LIN {X 0,Y 141.13,Z 751.048,A -85,B 0,C 180,E1 27006.176,E2 27006.176} C_VEL
LIN {X 0,Y 135.268,Z 754.68,A -85,B 0,C 180,E1 27012.954,E2 27012.954} C_VEL
LIN {X 0,Y 132.366,Z 756.637,A -85,B 0,C 180,E1 27014.356,E2 27014.356} C_VEL
LIN {X 0,Y 102.125,Z 773.9,A -85,B 0,C 180,E1 27021.98,E2 27021.98} C_VEL
LIN {X 0,Y 74.272,Z 785.098,A -85,B 0,C 180,E1 27035.392,E2 27035.392} C_VEL
LIN {X 0,Y 55.149,Z 790.593,A -85,B 0,C 180,E1 27056.715,E2 27056.715} C_VEL
LIN {X 0,Y 47.188,Z 792.386,A -85,B 0,C 180,E1 27090.017,E2 27090.017} C_VEL
LIN {X 0,Y 55.18,Z 790.549,A -85,B 0,C 180,E1 27123.299,E2 27123.299} C_VEL
LIN {X 0,Y 80.125,Z 782.969,A -85,B 0,C 180,E1 27148.264,E2 27148.264} C_VEL
LIN {X 0,Y 109.212,Z 770.247,A -85,B 0,C 180,E1 27160.115,E2 27160.115} C_VEL
LIN {X 0,Y 134.009,Z 755.358,A -85,B 0,C 180,E1 27165.896,E2 27165.896} C_VEL
LIN {X 0,Y 138.304,Z 752.387,A -85,B 0,C 180,E1 27170.176,E2 27170.176} C_VEL
LIN {X 0,Y 141.523,Z 750.747,A -85,B 0,C 180,E1 27175.02,E2 27175.02} C_VEL
LIN {X 0,Y 143.867,Z 750.723,A -85,B 0,C 180,E1 27180.669,E2 27180.669} C_VEL
LIN {X 0,Y 142.079,Z 752.687,A -85,B 0,C 180,E1 27182.028,E2 27182.028} C_VEL
LIN {X 0,Y 110.658,Z 774.445,A -85,B 0,C 180,E1 27187.223,E2 27187.223} C_VEL
LIN {X 0,Y 84.426,Z 788.358,A -85,B 0,C 180,E1 27195.358,E2 27195.358} C_VEL
LIN {X 0,Y 72.954,Z 792.741,A -85,B 0,C 180,E1 27198.842,E2 27198.842} C_VEL
LIN {X 0,Y 55.265,Z 797.756,A -85,B 0,C 180,E1 27205.481,E2 27205.481} C_VEL
LIN {X 0,Y 53.646,Z 798.256,A -85,B 0,C 180,E1 27206.938,E2 27206.938} C_VEL
LIN {X 0,Y 36.915,Z 804.117,A -85,B 0,C 180,E1 27245.763,E2 27245.763} C_VEL
LIN {X 0,Y 36.814,Z 805.147,A -85,B 0,C 180,E1 27269.978,E2 27269.978} C_VEL
LIN {X 0,Y 42.3,Z 802.077,A -85,B 0,C 180,E1 27315.686,E2 27315.686} C_VEL
LIN {X 0,Y 70.517,Z 792.25,A -85,B 0,C 180,E1 27345.009,E2 27345.009} C_VEL
LIN {X 0,Y 104.257,Z 776.595,A -85,B 0,C 180,E1 27355.878,E2 27355.878} C_VEL
LIN {X 0,Y 136.258,Z 756.023,A -85,B 0,C 180,E1 27360.693,E2 27360.693} C_VEL
LIN {X 0,Y 136.347,Z 755.474,A -85,B 0,C 180,E1 27362.184,E2 27362.184} C_VEL
LIN {X 0,Y 133.996,Z 756.111,A -85,B 0,C 180,E1 27366.506,E2 27366.506} C_VEL
LIN {X 0,Y 130.445,Z 758.02,A -85,B 0,C 180,E1 27370.436,E2 27370.436} C_VEL
LIN {X 0,Y 126.009,Z 760.827,A -85,B 0,C 180,E1 27371.835,E2 27371.835} C_VEL
LIN {X 0,Y 95.969,Z 776.64,A -85,B 0,C 180,E1 27378.841,E2 27378.841} C_VEL
LIN {X 0,Y 70.035,Z 786.286,A -85,B 0,C 180,E1 27390.172,E2 27390.172} C_VEL
LIN {X 0,Y 48.81,Z 791.778,A -85,B 0,C 180,E1 27411.678,E2 27411.678} C_VEL
LIN {X 0,Y 39.399,Z 793.569,A -85,B 0,C 180,E1 27450.02,E2 27450.02} C_VEL
LIN {X 0,Y 48.842,Z 791.735,A -85,B 0,C 180,E1 27488.334,E2 27488.334} C_VEL
LIN {X 0,Y 73.154,Z 785.238,A -85,B 0,C 180,E1 27511.616,E2 27511.616} C_VEL
LIN {X 0,Y 103.958,Z 772.802,A -85,B 0,C 180,E1 27523.35,E2 27523.35} C_VEL
LIN {X 0,Y 128.144,Z 759.249,A -85,B 0,C 180,E1 27528.457,E2 27528.457} C_VEL
LIN {X 0,Y 132.081,Z 756.912,A -85,B 0,C 180,E1 27531.11,E2 27531.11} C_VEL
LIN {X 0,Y 135.125,Z 755.518,A -85,B 0,C 180,E1 27535.552,E2 27535.552} C_VEL
LIN {X 0,Y 136.285,Z 755.805,A -85,B 0,C 180,E1 27539.325,E2 27539.325} C_VEL
LIN {X 0,Y 104.245,Z 776.442,A -85,B 0,C 180,E1 27544.079,E2 27544.079} C_VEL
LIN {X 0,Y 70.536,Z 792.156,A -85,B 0,C 180,E1 27554.96,E2 27554.96} C_VEL
LIN {X 0,Y 53.646,Z 798.256,A -85,B 0,C 180,E1 27566.938,E2 27566.938} C_VEL
LIN {X 0,Y 39.847,Z 801.381,A -85,B 0,C 180,E1 27579.711,E2 27579.711} C_VEL
LIN {X 0,Y 29.106,Z 803.028,A -85,B 0,C 180,E1 27603.278,E2 27603.278} C_VEL
LIN {X 0,Y 28.825,Z 803.933,A -85,B 0,C 180,E1 27629.972,E2 27629.972} C_VEL
LIN {X 0,Y 37.05,Z 800.835,A -85,B 0,C 180,E1 27684.776,E2 27684.776} C_VEL
LIN {X 0,Y 68.847,Z 790.999,A -85,B 0,C 180,E1 27711.647,E2 27711.647} C_VEL
LIN {X 0,Y 103.388,Z 775.666,A -85,B 0,C 180,E1 27720.281,E2 27720.281} C_VEL
LIN {X 0,Y 127.008,Z 761.504,A -85,B 0,C 180,E1 27723.22,E2 27723.22} C_VEL
LIN {X 0,Y 128.828,Z 760.178,A -85,B 0,C 180,E1 27723.807,E2 27723.807} C_VEL
LIN {X 0,Y 125.265,Z 761.647,A -85,B 0,C 180,E1 27728.171,E2 27728.171} C_VEL
LIN {X 0,Y 93.737,Z 777.832,A -85,B 0,C 180,E1 27734.315,E2 27734.315} C_VEL
LIN {X 0,Y 66.45,Z 787.475,A -85,B 0,C 180,E1 27744.334,E2 27744.334} C_VEL
LIN {X 0,Y 42.946,Z 792.966,A -85,B 0,C 180,E1 27765.19,E2 27765.19} C_VEL
LIN {X 0,Y 31.589,Z 794.756,A -85,B 0,C 180,E1 27810.025,E2 27810.025} C_VEL
LIN {X 0,Y 44.361,Z 792.68,A -85,B 0,C 180,E1 27856.879,E2 27856.879} C_VEL
LIN {X 0,Y 73.104,Z 785.355,A -85,B 0,C 180,E1 27878.774,E2 27878.774} C_VEL
LIN {X 0,Y 105.693,Z 772.261,A -85,B 0,C 180,E1 27888.307,E2 27888.307} C_VEL
LIN {X 0,Y 125.28,Z 761.436,A -85,B 0,C 180,E1 27891.786,E2 27891.786} C_VEL
LIN {X 0,Y 128.816,Z 759.994,A -85,B 0,C 180,E1 27896.178,E2 27896.178} C_VEL
LIN {X 0,Y 109.807,Z 771.944,A -85,B 0,C 180,E1 27898.744,E2 27898.744} C_VEL
LIN {X 0,Y 76.098,Z 788.137,A -85,B 0,C 180,E1 27905.75,E2 27905.75} C_VEL
LIN {X 0,Y 48.423,Z 797.618,A -85,B 0,C 180,E1 27920.311,E2 27920.311} C_VEL
LIN {X 0,Y 29.106,Z 803.028,A -85,B 0,C 180,E1 27963.278,E2 27963.278} C_VEL
LIN {X 0,Y 26.216,Z 803.383,A -85,B 0,C 180,E1 27980.281,E2 27980.281} C_VEL
LIN {X 0,Y 26.217,Z 800.978,A -85,B 0,C 180,E1 28042.764,E2 28042.764} C_VEL
LIN {X 0,Y 56.12,Z 793.66,A -85,B 0,C 180,E1 28074.433,E2 28074.433} C_VEL
LIN {X 0,Y 90.97,Z 780.586,A -85,B 0,C 180,E1 28083.207,E2 28083.207} C_VEL
LIN {X 0,Y 113.201,Z 769.259,A -85,B 0,C 180,E1 28085.73,E2 28085.73} C_VEL
LIN {X 0,Y 81.265,Z 783.16,A -85,B 0,C 180,E1 28092.058,E2 28092.058} C_VEL
LIN {X 0,Y 50.114,Z 791.904,A -85,B 0,C 180,E1 28105.032,E2 28105.032} C_VEL
LIN {X 0,Y 28.183,Z 795.415,A -85,B 0,C 180,E1 28137.54,E2 28137.54} C_VEL
LIN {X 0,Y 28.206,Z 795.39,A -85,B 0,C 180,E1 28202.498,E2 28202.498} C_VEL
LIN {X 0,Y 56.821,Z 790.364,A -85,B 0,C 180,E1 28238.881,E2 28238.881} C_VEL
LIN {X 0,Y 88.526,Z 780.33,A -85,B 0,C 180,E1 28249.594,E2 28249.594} C_VEL
LIN {X 0,Y 113.197,Z 769.09,A -85,B 0,C 180,E1 28254.216,E2 28254.216} C_VEL
LIN {X 0,Y 79.519,Z 785.367,A -85,B 0,C 180,E1 28258.743,E2 28258.743} C_VEL
LIN {X 0,Y 46.237,Z 796.364,A -85,B 0,C 180,E1 28270.691,E2 28270.691} C_VEL
LIN {X 0,Y 21.523,Z 801.927,A -85,B 0,C 180,E1 28318.32,E2 28318.32} C_VEL
LIN {X 0,Y 20.825,Z 802.718,A -85,B 0,C 180,E1 28349.962,E2 28349.962} C_VEL
LIN {X 0,Y 26.217,Z 800.978,A -85,B 0,C 180,E1 28402.764,E2 28402.764} C_VEL
LIN {X 0,Y 33.884,Z 798.843,A -85,B 0,C 180,E1 28422.95,E2 28422.95} C_VEL
LIN {X 0,Y 48.682,Z 794.374,A -85,B 0,C 180,E1 28440.59,E2 28440.59} C_VEL
LIN {X 0,Y 50.712,Z 793.84,A -85,B 0,C 180,E1 28441.362,E2 28441.362} C_VEL
LIN {X 0,Y 76.198,Z 785.741,A -85,B 0,C 180,E1 28446.637,E2 28446.637} C_VEL
LIN {X 0,Y 76.303,Z 785.609,A -85,B 0,C 180,E1 28447.283,E2 28447.283} C_VEL
LIN {X 0,Y 47.344,Z 793.089,A -85,B 0,C 180,E1 28456.449,E2 28456.449} C_VEL
LIN {X 0,Y 22.001,Z 796.601,A -85,B 0,C 180,E1 28486.566,E2 28486.566} C_VEL
LIN {X 0,Y 22.027,Z 796.576,A -85,B 0,C 180,E1 28573.47,E2 28573.47} C_VEL
LIN {X 0,Y 54.647,Z 791.518,A -85,B 0,C 180,E1 28606.631,E2 28606.631} C_VEL
LIN {X 0,Y 76.341,Z 785.486,A -85,B 0,C 180,E1 28612.66,E2 28612.66} C_VEL
LIN {X 0,Y 73.357,Z 786.71,A -85,B 0,C 180,E1 28613.712,E2 28613.712} C_VEL
LIN {X 0,Y 37.959,Z 796.821,A -85,B 0,C 180,E1 28624.055,E2 28624.055} C_VEL
LIN {X 0,Y 17.803,Z 800.424,A -85,B 0,C 180,E1 28651.658,E2 28651.658} C_VEL
LIN {X 0,Y 12.836,Z 801.505,A -85,B 0,C 180,E1 28709.938,E2 28709.938} C_VEL
LIN {X 0,Y 30.675,Z 798.349,A -85,B 0,C 180,E1 28790.64,E2 28790.64} C_VEL
LIN {X 0,Y 50.712,Z 793.84,A -85,B 0,C 180,E1 28801.362,E2 28801.362} C_VEL
LIN {X 0,Y 47.229,Z 794.189,A -85,B 0,C 180,E1 28805.113,E2 28805.113} C_VEL
LIN {X 0,Y 18.1,Z 797.697,A -85,B 0,C 180,E1 28826.556,E2 28826.556} C_VEL
LIN {X 0,Y 17.221,Z 797.762,A -85,B 0,C 180,E1 28951.638,E2 28951.638} C_VEL
LIN {X 0,Y 31.108,Z 796.48,A -85,B 0,C 180,E1 28966.867,E2 28966.867} C_VEL
LIN {X 0,Y 36.979,Z 795.832,A -85,B 0,C 180,E1 28971.997,E2 28971.997} C_VEL
LIN {X 0,Y 15.203,Z 799.19,A -85,B 0,C 180,E1 28984.607,E2 28984.607} C_VEL
LIN {X 0,Y 4.811,Z 800.285,A -85,B 0,C 180,E1 29069.834,E2 29069.834} C_VEL
LIN {X 0,Y 30.434,Z 797.108,A -85,B 0,C 180,E1 29166.009,E2 29166.009} C_VEL
LIN {X 0,Y 36.911,Z 795.896,A -85,B 0,C 180,E1 29167.955,E2 29167.955} C_VEL
LIN {X 0,Y 31.072,Z 796.524,A -85,B 0,C 180,E1 29173.079,E2 29173.079} C_VEL
LIN {X 0,Y 18.1,Z 797.697,A -85,B 0,C 180,E1 29186.556,E2 29186.556} C_VEL
LIN {X 0,Y 16.552,Z 799.69,A -85,B 0,C 180,E1 29189.815,E2 29189.815} C_VEL
LIN {X 0,Y 16.552,Z 875,A -85,B 0,C 180,E1 29189.815,E2 29189.815} C_VEL
LIN {X 0,Y 16.552,Z 875,A -85,B 0,C 180,E1 29189.815,E2 29189.815}

QRS_NEXT_CUT()
PTP {E1 29336.944,E2 29336.944}
PTP {X 0,Y 607.85,A -85,B 0,C 180,E1 29336.944,E2 29336.944,E3 0,E4 0,E5 0,E6 0}
QRS_SPEED_INIT()
LIN {X 0,Y 607.85,Z 875,A -85,B 0,C 180,E1 29336.944,E2 29336.944,E3 0,E4 0,E5 0,E6 0} C_VEL
LIN {X 0,Y 607.85,Z 296.842,A -85,B 0,C 180,E1 29336.944,E2 29336.944} C_VEL
LIN {X 0,Y 607.85,Z 288.764,A -85,B 0,C 180,E1 29336.944,E2 29336.944} C_VEL
LIN {X 0,Y 607.871,Z 286.764,A -85,B 0,C 180,E1 29336.755,E2 29336.755} C_VEL
LIN {X 0,Y 607.835,Z 286.764,A -85,B 0,C 180,E1 29333.672,E2 29333.672} C_VEL
LIN {X 0,Y 607.851,Z 286.764,A -85,B 0,C 180,E1 29330.914,E2 29330.914} C_VEL
LIN {X 0,Y 607.842,Z 286.764,A -85,B 0,C 180,E1 29327.652,E2 29327.652} C_VEL
LIN {X 0,Y 607.86,Z 286.764,A -85,B 0,C 180,E1 29324.839,E2 29324.839} C_VEL
LIN {X 0,Y 607.85,Z 286.762,A -85,B 0,C 180,E1 29321.589,E2 29321.589} C_VEL
LIN {X 0,Y 607.875,Z 286.764,A -85,B 0,C 180,E1 29318.684,E2 29318.684} C_VEL
LIN {X 0,Y 607.856,Z 286.761,A -85,B 0,C 180,E1 29315.511,E2 29315.511} C_VEL
LIN {X 0,Y 607.886,Z 286.764,A -85,B 0,C 180,E1 29312.577,E2 29312.577} C_VEL
LIN {X 0,Y 607.862,Z 286.761,A -85,B 0,C 180,E1 29309.451,E2 29309.451} C_VEL
LIN {X 0,Y 607.899,Z 286.764,A -85,B 0,C 180,E1 29306.451,E2 29306.451} C_VEL
LIN {X 0,Y 607.865,Z 286.76,A -85,B 0,C 180,E1 29303.338,E2 29303.338} C_VEL
LIN {X 0,Y 607.909,Z 286.765,A -85,B 0,C 180,E1 29300.329,E2 29300.329} C_VEL
LIN {X 0,Y 607.867,Z 286.76,A -85,B 0,C 180,E1 29297.188,E2 29297.188} C_VEL
LIN {X 0,Y 607.915,Z 286.761,A -85,B 0,C 180,E1 29294.083,E2 29294.083} C_VEL
LIN {X 0,Y 607.87,Z 286.76,A -85,B 0,C 180,E1 29290.975,E2 29290.975} C_VEL
LIN {X 0,Y 607.912,Z 286.759,A -85,B 0,C 180,E1 29287.841,E2 29287.841} C_VEL
LIN {X 0,Y 607.879,Z 286.761,A -85,B 0,C 180,E1 29284.687,E2 29284.687} C_VEL
LIN {X 0,Y 607.911,Z 286.755,A -85,B 0,C 180,E1 29281.535,E2 29281.535} C_VEL
LIN {X 0,Y 607.905,Z 286.765,A -85,B 0,C 180,E1 29278.273,E2 29278.273} C_VEL
LIN {X 0,Y 607.909,Z 287.028,A -85,B 0,C 180,E1 29276.259,E2 29276.259} C_VEL
LIN {X 0,Y 607.912,Z 319.926,A -85,B 0,C 180,E1 29273.454,E2 29273.454} C_VEL
LIN {X 0,Y 607.914,Z 334.281,A -85,B 0,C 180,E1 29272.278,E2 29272.278} C_VEL
LIN {X 0,Y 607.916,Z 541.958,A -85,B 0,C 180,E1 29269.666,E2 29269.666} C_VEL
LIN {X 0,Y 607.911,Z 560.928,A -85,B 0,C 180,E1 29269.25,E2 29269.25} C_VEL
LIN {X 0,Y 607.902,Z 579.266,A -85,B 0,C 180,E1 29268.668,E2 29268.668} C_VEL
LIN {X 0,Y 607.897,Z 597.163,A -85,B 0,C 180,E1 29267.913,E2 29267.913} C_VEL
LIN {X 0,Y 607.919,Z 613.869,A -85,B 0,C 180,E1 29267.023,E2 29267.023} C_VEL
LIN {X 0,Y 607.917,Z 629.704,A -85,B 0,C 180,E1 29265.991,E2 29265.991} C_VEL
LIN {X 0,Y 607.917,Z 644.611,A -85,B 0,C 180,E1 29264.818,E2 29264.818} C_VEL
LIN {X 0,Y 607.915,Z 658.52,A -85,B 0,C 180,E1 29263.506,E2 29263.506} C_VEL
LIN {X 0,Y 607.917,Z 671.323,A -85,B 0,C 180,E1 29262.056,E2 29262.056} C_VEL
LIN {X 0,Y 607.911,Z 682.566,A -85,B 0,C 180,E1 29260.519,E2 29260.519} C_VEL
LIN {X 0,Y 607.914,Z 692.264,A -85,B 0,C 180,E1 29258.894,E2 29258.894} C_VEL
LIN {X 0,Y 607.911,Z 699.987,A -85,B 0,C 180,E1 29257.276,E2 29257.276} C_VEL
LIN {X 0,Y 607.907,Z 706.267,A -85,B 0,C 180,E1 29255.569,E2 29255.569} C_VEL
LIN {X 0,Y 607.918,Z 710.775,A -85,B 0,C 180,E1 29253.867,E2 29253.867} C_VEL
LIN {X 0,Y 607.917,Z 713.734,A -85,B 0,C 180,E1 29252.074,E2 29252.074} C_VEL
LIN {X 0,Y 607.908,Z 714.929,A -85,B 0,C 180,E1 29250.283,E2 29250.283} C_VEL
LIN {X 0,Y 607.915,Z 714.38,A -85,B 0,C 180,E1 29248.492,E2 29248.492} C_VEL
LIN {X 0,Y 607.909,Z 712.08,A -85,B 0,C 180,E1 29246.7,E2 29246.7} C_VEL
LIN {X 0,Y 607.914,Z 708.217,A -85,B 0,C 180,E1 29244.999,E2 29244.999} C_VEL
LIN {X 0,Y 607.91,Z 702.635,A -85,B 0,C 180,E1 29243.294,E2 29243.294} C_VEL
LIN {X 0,Y 607.917,Z 695.641,A -85,B 0,C 180,E1 29241.678,E2 29241.678} C_VEL
LIN {X 0,Y 607.913,Z 686.781,A -85,B 0,C 180,E1 29240.056,E2 29240.056} C_VEL
LIN {X 0,Y 607.917,Z 676.477,A -85,B 0,C 180,E1 29238.521,E2 29238.521} C_VEL
LIN {X 0,Y 607.913,Z 664.743,A -85,B 0,C 180,E1 29237.075,E2 29237.075} C_VEL
LIN {X 0,Y 607.917,Z 651.561,A -85,B 0,C 180,E1 29235.718,E2 29235.718} C_VEL
LIN {X 0,Y 607.917,Z 636.801,A -85,B 0,C 180,E1 29234.45,E2 29234.45} C_VEL
LIN {X 0,Y 607.917,Z 620.944,A -85,B 0,C 180,E1 29233.322,E2 29233.322} C_VEL
LIN {X 0,Y 607.902,Z 603.949,A -85,B 0,C 180,E1 29232.335,E2 29232.335} C_VEL
LIN {X 0,Y 607.918,Z 586.961,A -85,B 0,C 180,E1 29231.543,E2 29231.543} C_VEL
LIN {X 0,Y 607.909,Z 569.084,A -85,B 0,C 180,E1 29230.895,E2 29230.895} C_VEL
LIN {X 0,Y 607.915,Z 550.763,A -85,B 0,C 180,E1 29230.413,E2 29230.413} C_VEL
LIN {X 0,Y 607.918,Z 531.813,A -85,B 0,C 180,E1 29230.096,E2 29230.096} C_VEL
LIN {X 0,Y 607.91,Z 334.059,A -85,B 0,C 180,E1 29227.621,E2 29227.621} C_VEL
LIN {X 0,Y 607.918,Z 296.429,A -85,B 0,C 180,E1 29224.475,E2 29224.475} C_VEL
LIN {X 0,Y 607.909,Z 286.947,A -85,B 0,C 180,E1 29223.636,E2 29223.636} C_VEL
LIN {X 0,Y 607.91,Z 286.756,A -85,B 0,C 180,E1 29220.543,E2 29220.543} C_VEL
LIN {X 0,Y 607.889,Z 286.762,A -85,B 0,C 180,E1 29217.352,E2 29217.352} C_VEL
LIN {X 0,Y 607.91,Z 286.758,A -85,B 0,C 180,E1 29214.181,E2 29214.181} C_VEL
LIN {X 0,Y 607.877,Z 286.76,A -85,B 0,C 180,E1 29211.075,E2 29211.075} C_VEL
LIN {X 0,Y 607.91,Z 286.76,A -85,B 0,C 180,E1 29207.98,E2 29207.98} C_VEL
LIN {X 0,Y 607.872,Z 286.759,A -85,B 0,C 180,E1 29204.882,E2 29204.882} C_VEL
LIN {X 0,Y 607.918,Z 286.764,A -85,B 0,C 180,E1 29201.696,E2 29201.696} C_VEL
LIN {X 0,Y 607.877,Z 286.759,A -85,B 0,C 180,E1 29198.565,E2 29198.565} C_VEL
LIN {X 0,Y 607.879,Z 286.763,A -85,B 0,C 180,E1 29195.264,E2 29195.264} C_VEL
LIN {X 0,Y 607.897,Z 286.758,A -85,B 0,C 180,E1 29192.203,E2 29192.203} C_VEL
LIN {X 0,Y 607.862,Z 286.762,A -85,B 0,C 180,E1 29189.028,E2 29189.028} C_VEL
LIN {X 0,Y 607.903,Z 286.759,A -85,B 0,C 180,E1 29186.05,E2 29186.05} C_VEL
LIN {X 0,Y 607.854,Z 286.763,A -85,B 0,C 180,E1 29182.91,E2 29182.91} C_VEL
LIN {X 0,Y 607.905,Z 286.76,A -85,B 0,C 180,E1 29179.905,E2 29179.905} C_VEL
LIN {X 0,Y 607.846,Z 286.763,A -85,B 0,C 180,E1 29176.801,E2 29176.801} C_VEL
LIN {X 0,Y 607.909,Z 286.761,A -85,B 0,C 180,E1 29173.798,E2 29173.798} C_VEL
LIN {X 0,Y 607.839,Z 286.764,A -85,B 0,C 180,E1 29170.713,E2 29170.713} C_VEL
LIN {X 0,Y 607.899,Z 286.762,A -85,B 0,C 180,E1 29167.751,E2 29167.751} C_VEL
LIN {X 0,Y 607.834,Z 286.764,A -85,B 0,C 180,E1 29164.718,E2 29164.718} C_VEL
LIN {X 0,Y 607.866,Z 286.764,A -85,B 0,C 180,E1 29161.885,E2 29161.885} C_VEL
LIN {X 0,Y 607.834,Z 286.765,A -85,B 0,C 180,E1 29158.775,E2 29158.775} C_VEL
LIN {X 0,Y 607.846,Z 286.764,A -85,B 0,C 180,E1 29156.039,E2 29156.039} C_VEL
LIN {X 0,Y 607.848,Z 286.763,A -85,B 0,C 180,E1 29152.819,E2 29152.819} C_VEL
LIN {X 0,Y 607.847,Z 286.764,A -85,B 0,C 180,E1 29150.054,E2 29150.054} C_VEL
LIN {X 0,Y 607.857,Z 286.762,A -85,B 0,C 180,E1 29146.783,E2 29146.783} C_VEL
LIN {X 0,Y 607.856,Z 286.764,A -85,B 0,C 180,E1 29143.958,E2 29143.958} C_VEL
LIN {X 0,Y 607.861,Z 286.761,A -85,B 0,C 180,E1 29140.694,E2 29140.694} C_VEL
LIN {X 0,Y 607.873,Z 286.764,A -85,B 0,C 180,E1 29137.771,E2 29137.771} C_VEL
LIN {X 0,Y 607.862,Z 286.761,A -85,B 0,C 180,E1 29134.557,E2 29134.557} C_VEL
LIN {X 0,Y 607.889,Z 286.764,A -85,B 0,C 180,E1 29131.618,E2 29131.618} C_VEL
LIN {X 0,Y 607.865,Z 286.76,A -85,B 0,C 180,E1 29128.432,E2 29128.432} C_VEL
LIN {X 0,Y 607.918,Z 286.763,A -85,B 0,C 180,E1 29125.314,E2 29125.314} C_VEL
LIN {X 0,Y 607.867,Z 286.76,A -85,B 0,C 180,E1 29122.274,E2 29122.274} C_VEL
LIN {X 0,Y 607.914,Z 286.761,A -85,B 0,C 180,E1 29119.162,E2 29119.162} C_VEL
LIN {X 0,Y 607.871,Z 286.76,A -85,B 0,C 180,E1 29116.042,E2 29116.042} C_VEL
LIN {X 0,Y 607.913,Z 286.759,A -85,B 0,C 180,E1 29112.914,E2 29112.914} C_VEL
LIN {X 0,Y 607.88,Z 286.761,A -85,B 0,C 180,E1 29109.778,E2 29109.778} C_VEL
LIN {X 0,Y 607.908,Z 286.756,A -85,B 0,C 180,E1 29106.54,E2 29106.54} C_VEL
LIN {X 0,Y 607.897,Z 286.884,A -85,B 0,C 180,E1 29103.498,E2 29103.498} C_VEL
LIN {X 0,Y 607.908,Z 287.709,A -85,B 0,C 180,E1 29103.382,E2 29103.382} C_VEL
LIN {X 0,Y 607.913,Z 340.141,A -85,B 0,C 180,E1 29100.435,E2 29100.435} C_VEL
LIN {X 0,Y 607.885,Z 390.509,A -85,B 0,C 180,E1 29097.701,E2 29097.701} C_VEL
LIN {X 0,Y 607.913,Z 616.116,A -85,B 0,C 180,E1 29094.784,E2 29094.784} C_VEL
LIN {X 0,Y 607.918,Z 653.733,A -85,B 0,C 180,E1 29094.278,E2 29094.278} C_VEL
LIN {X 0,Y 607.906,Z 673.698,A -85,B 0,C 180,E1 29093.84,E2 29093.84} C_VEL
LIN {X 0,Y 607.911,Z 693.06,A -85,B 0,C 180,E1 29093.249,E2 29093.249} C_VEL
LIN {X 0,Y 607.915,Z 712.501,A -85,B 0,C 180,E1 29092.482,E2 29092.482} C_VEL
LIN {X 0,Y 607.919,Z 731.168,A -85,B 0,C 180,E1 29091.567,E2 29091.567} C_VEL
LIN {X 0,Y 607.917,Z 749.766,A -85,B 0,C 180,E1 29090.456,E2 29090.456} C_VEL
LIN {X 0,Y 607.913,Z 767.254,A -85,B 0,C 180,E1 29089.204,E2 29089.204} C_VEL
LIN {X 0,Y 607.911,Z 783.162,A -85,B 0,C 180,E1 29087.863,E2 29087.863} C_VEL
LIN {X 0,Y 607.915,Z 797.673,A -85,B 0,C 180,E1 29086.432,E2 29086.432} C_VEL
LIN {X 0,Y 607.909,Z 811.263,A -85,B 0,C 180,E1 29084.867,E2 29084.867} C_VEL
LIN {X 0,Y 607.918,Z 823.719,A -85,B 0,C 180,E1 29083.176,E2 29083.176} C_VEL
LIN {X 0,Y 607.906,Z 834.252,A -85,B 0,C 180,E1 29081.479,E2 29081.479} C_VEL
LIN {X 0,Y 607.907,Z 843.561,A -85,B 0,C 180,E1 29079.658,E2 29079.658} C_VEL
LIN {X 0,Y 607.907,Z 850.973,A -85,B 0,C 180,E1 29077.846,E2 29077.846} C_VEL
LIN {X 0,Y 607.913,Z 856.989,A -85,B 0,C 180,E1 29075.947,E2 29075.947} C_VEL
LIN {X 0,Y 607.913,Z 861.292,A -85,B 0,C 180,E1 29074.055,E2 29074.055} C_VEL
LIN {X 0,Y 607.909,Z 863.95,A -85,B 0,C 180,E1 29072.168,E2 29072.168} C_VEL
LIN {X 0,Y 607.902,Z 864.94,A -85,B 0,C 180,E1 29070.283,E2 29070.283} C_VEL
LIN {X 0,Y 607.904,Z 864.372,A -85,B 0,C 180,E1 29068.398,E2 29068.398} C_VEL
LIN {X 0,Y 607.908,Z 862.082,A -85,B 0,C 180,E1 29066.417,E2 29066.417} C_VEL
LIN {X 0,Y 607.91,Z 858.255,A -85,B 0,C 180,E1 29064.526,E2 29064.526} C_VEL
LIN {X 0,Y 607.913,Z 852.689,A -85,B 0,C 180,E1 29062.629,E2 29062.629} C_VEL
LIN {X 0,Y 607.919,Z 845.655,A -85,B 0,C 180,E1 29060.82,E2 29060.82} C_VEL
LIN {X 0,Y 607.909,Z 836.843,A -85,B 0,C 180,E1 29059.001,E2 29059.001} C_VEL
LIN {X 0,Y 607.911,Z 826.516,A -85,B 0,C 180,E1 29057.247,E2 29057.247} C_VEL
LIN {X 0,Y 607.917,Z 815.136,A -85,B 0,C 180,E1 29055.62,E2 29055.62} C_VEL
LIN {X 0,Y 607.91,Z 801.355,A -85,B 0,C 180,E1 29053.96,E2 29053.96} C_VEL
LIN {X 0,Y 607.918,Z 785.904,A -85,B 0,C 180,E1 29052.385,E2 29052.385} C_VEL
LIN {X 0,Y 607.913,Z 769.201,A -85,B 0,C 180,E1 29050.945,E2 29050.945} C_VEL
LIN {X 0,Y 607.917,Z 752.006,A -85,B 0,C 180,E1 29049.694,E2 29049.694} C_VEL
LIN {X 0,Y 607.919,Z 734.735,A -85,B 0,C 180,E1 29048.636,E2 29048.636} C_VEL
LIN {X 0,Y 607.909,Z 715.856,A -85,B 0,C 180,E1 29047.671,E2 29047.671} C_VEL
LIN {X 0,Y 607.907,Z 696.731,A -85,B 0,C 180,E1 29046.879,E2 29046.879} C_VEL
LIN {X 0,Y 607.906,Z 676.741,A -85,B 0,C 180,E1 29046.237,E2 29046.237} C_VEL
LIN {X 0,Y 607.917,Z 657.663,A -85,B 0,C 180,E1 29045.799,E2 29045.799} C_VEL
LIN {X 0,Y 607.913,Z 631.428,A -85,B 0,C 180,E1 29045.411,E2 29045.411} C_VEL
LIN {X 0,Y 607.88,Z 396.039,A -85,B 0,C 180,E1 29042.375,E2 29042.375} C_VEL
LIN {X 0,Y 607.887,Z 389.594,A -85,B 0,C 180,E1 29042.26,E2 29042.26} C_VEL
LIN {X 0,Y 607.918,Z 333.456,A -85,B 0,C 180,E1 29039.195,E2 29039.195} C_VEL
LIN {X 0,Y 607.905,Z 287.421,A -85,B 0,C 180,E1 29036.592,E2 29036.592} C_VEL
LIN {X 0,Y 607.894,Z 286.812,A -85,B 0,C 180,E1 29036.452,E2 29036.452} C_VEL
LIN {X 0,Y 607.917,Z 286.756,A -85,B 0,C 180,E1 29033.343,E2 29033.343} C_VEL
LIN {X 0,Y 607.877,Z 286.76,A -85,B 0,C 180,E1 29030.099,E2 29030.099} C_VEL
LIN {X 0,Y 607.911,Z 286.761,A -85,B 0,C 180,E1 29026.957,E2 29026.957} C_VEL
LIN {X 0,Y 607.872,Z 286.76,A -85,B 0,C 180,E1 29023.827,E2 29023.827} C_VEL
LIN {X 0,Y 607.914,Z 286.765,A -85,B 0,C 180,E1 29020.641,E2 29020.641} C_VEL
LIN {X 0,Y 607.88,Z 286.758,A -85,B 0,C 180,E1 29017.487,E2 29017.487} C_VEL
LIN {X 0,Y 607.873,Z 286.763,A -85,B 0,C 180,E1 29014.174,E2 29014.174} C_VEL
LIN {X 0,Y 607.903,Z 286.758,A -85,B 0,C 180,E1 29011.095,E2 29011.095} C_VEL
LIN {X 0,Y 607.86,Z 286.762,A -85,B 0,C 180,E1 29007.956,E2 29007.956} C_VEL
LIN {X 0,Y 607.92,Z 286.759,A -85,B 0,C 180,E1 29004.901,E2 29004.901} C_VEL
LIN {X 0,Y 607.852,Z 286.762,A -85,B 0,C 180,E1 29001.823,E2 29001.823} C_VEL
LIN {X 0,Y 607.918,Z 286.762,A -85,B 0,C 180,E1 28998.706,E2 28998.706} C_VEL
LIN {X 0,Y 607.845,Z 286.763,A -85,B 0,C 180,E1 28995.65,E2 28995.65} C_VEL
LIN {X 0,Y 607.919,Z 286.764,A -85,B 0,C 180,E1 28992.539,E2 28992.539} C_VEL
LIN {X 0,Y 607.839,Z 286.763,A -85,B 0,C 180,E1 28989.563,E2 28989.563} C_VEL
LIN {X 0,Y 607.916,Z 286.764,A -85,B 0,C 180,E1 28986.516,E2 28986.516} C_VEL
LIN {X 0,Y 607.833,Z 286.764,A -85,B 0,C 180,E1 28983.489,E2 28983.489} C_VEL
LIN {X 0,Y 607.913,Z 286.765,A -85,B 0,C 180,E1 28980.471,E2 28980.471} C_VEL
LIN {X 0,Y 607.826,Z 286.765,A -85,B 0,C 180,E1 28977.454,E2 28977.454} C_VEL
LIN {X 0,Y 607.871,Z 286.764,A -85,B 0,C 180,E1 28976.755,E2 28976.755} C_VEL
LIN {X 0,Y 606.936,Z 286.888,A -85,B 0,C 180,E1 28976.029,E2 28976.029} C_VEL
LIN {X 0,Y 600.437,Z 287.691,A -85,B 0,C 180,E1 28973.992,E2 28973.992} C_VEL
LIN {X 0,Y 599.891,Z 287.754,A -85,B 0,C 180,E1 28973.462,E2 28973.462} C_VEL
LIN {X 0,Y 599.962,Z 287.753,A -85,B 0,C 180,E1 28970.503,E2 28970.503} C_VEL
LIN {X 0,Y 599.897,Z 287.753,A -85,B 0,C 180,E1 28967.486,E2 28967.486} C_VEL
LIN {X 0,Y 599.958,Z 287.752,A -85,B 0,C 180,E1 28964.535,E2 28964.535} C_VEL
LIN {X 0,Y 599.905,Z 287.751,A -85,B 0,C 180,E1 28961.437,E2 28961.437} C_VEL
LIN {X 0,Y 599.97,Z 287.754,A -85,B 0,C 180,E1 28958.389,E2 28958.389} C_VEL
LIN {X 0,Y 599.91,Z 287.75,A -85,B 0,C 180,E1 28955.27,E2 28955.27} C_VEL
LIN {X 0,Y 599.979,Z 287.75,A -85,B 0,C 180,E1 28952.185,E2 28952.185} C_VEL
LIN {X 0,Y 599.916,Z 287.751,A -85,B 0,C 180,E1 28949.114,E2 28949.114} C_VEL
LIN {X 0,Y 599.976,Z 287.749,A -85,B 0,C 180,E1 28946.063,E2 28946.063} C_VEL
LIN {X 0,Y 599.922,Z 287.751,A -85,B 0,C 180,E1 28942.968,E2 28942.968} C_VEL
LIN {X 0,Y 599.969,Z 287.747,A -85,B 0,C 180,E1 28939.838,E2 28939.838} C_VEL
LIN {X 0,Y 599.934,Z 287.751,A -85,B 0,C 180,E1 28936.743,E2 28936.743} C_VEL
LIN {X 0,Y 599.954,Z 287.745,A -85,B 0,C 180,E1 28933.493,E2 28933.493} C_VEL
LIN {X 0,Y 599.969,Z 287.755,A -85,B 0,C 180,E1 28930.285,E2 28930.285} C_VEL
LIN {X 0,Y 599.938,Z 287.748,A -85,B 0,C 180,E1 28927.106,E2 28927.106} C_VEL
LIN {X 0,Y 599.975,Z 287.752,A -85,B 0,C 180,E1 28924.051,E2 28924.051} C_VEL
LIN {X 0,Y 599.94,Z 287.748,A -85,B 0,C 180,E1 28920.874,E2 28920.874} C_VEL
LIN {X 0,Y 599.971,Z 287.752,A -85,B 0,C 180,E1 28917.707,E2 28917.707} C_VEL
LIN {X 0,Y 599.984,Z 288.004,A -85,B 0,C 180,E1 28916.553,E2 28916.553} C_VEL
LIN {X 0,Y 600.401,Z 291.081,A -85,B 0,C 180,E1 28916.24,E2 28916.24} C_VEL
LIN {X 0,Y 600.278,Z 327.914,A -85,B 0,C 180,E1 28913.095,E2 28913.095} C_VEL
LIN {X 0,Y 600.314,Z 334.297,A -85,B 0,C 180,E1 28912.575,E2 28912.575} C_VEL
LIN {X 0,Y 600.501,Z 346.221,A -85,B 0,C 180,E1 28912.404,E2 28912.404} C_VEL
LIN {X 0,Y 600.376,Z 542.325,A -85,B 0,C 180,E1 28909.917,E2 28909.917} C_VEL
LIN {X 0,Y 600.333,Z 561.284,A -85,B 0,C 180,E1 28909.493,E2 28909.493} C_VEL
LIN {X 0,Y 600.273,Z 579.732,A -85,B 0,C 180,E1 28908.896,E2 28908.896} C_VEL
LIN {X 0,Y 600.214,Z 597.173,A -85,B 0,C 180,E1 28908.15,E2 28908.15} C_VEL
LIN {X 0,Y 600.178,Z 613.876,A -85,B 0,C 180,E1 28907.249,E2 28907.249} C_VEL
LIN {X 0,Y 600.12,Z 629.709,A -85,B 0,C 180,E1 28906.204,E2 28906.204} C_VEL
LIN {X 0,Y 600.066,Z 644.618,A -85,B 0,C 180,E1 28905.016,E2 28905.016} C_VEL
LIN {X 0,Y 600.022,Z 658.526,A -85,B 0,C 180,E1 28903.687,E2 28903.687} C_VEL
LIN {X 0,Y 599.985,Z 671.33,A -85,B 0,C 180,E1 28902.218,E2 28902.218} C_VEL
LIN {X 0,Y 599.951,Z 682.571,A -85,B 0,C 180,E1 28900.66,E2 28900.66} C_VEL
LIN {X 0,Y 599.937,Z 692.268,A -85,B 0,C 180,E1 28899.013,E2 28899.013} C_VEL
LIN {X 0,Y 599.921,Z 699.99,A -85,B 0,C 180,E1 28897.373,E2 28897.373} C_VEL
LIN {X 0,Y 599.909,Z 706.269,A -85,B 0,C 180,E1 28895.643,E2 28895.643} C_VEL
LIN {X 0,Y 599.919,Z 710.778,A -85,B 0,C 180,E1 28893.918,E2 28893.918} C_VEL
LIN {X 0,Y 599.917,Z 713.736,A -85,B 0,C 180,E1 28892.101,E2 28892.101} C_VEL
LIN {X 0,Y 599.909,Z 714.929,A -85,B 0,C 180,E1 28890.286,E2 28890.286} C_VEL
LIN {X 0,Y 599.915,Z 714.38,A -85,B 0,C 180,E1 28888.472,E2 28888.472} C_VEL
LIN {X 0,Y 599.908,Z 712.08,A -85,B 0,C 180,E1 28886.656,E2 28886.656} C_VEL
LIN {X 0,Y 599.916,Z 708.216,A -85,B 0,C 180,E1 28884.932,E2 28884.932} C_VEL
LIN {X 0,Y 599.919,Z 702.634,A -85,B 0,C 180,E1 28883.204,E2 28883.204} C_VEL
LIN {X 0,Y 599.929,Z 695.639,A -85,B 0,C 180,E1 28881.567,E2 28881.567} C_VEL
LIN {X 0,Y 599.944,Z 686.779,A -85,B 0,C 180,E1 28879.922,E2 28879.922} C_VEL
LIN {X 0,Y 599.968,Z 676.473,A -85,B 0,C 180,E1 28878.367,E2 28878.367} C_VEL
LIN {X 0,Y 600,Z 664.738,A -85,B 0,C 180,E1 28876.901,E2 28876.901} C_VEL
LIN {X 0,Y 600.044,Z 651.243,A -85,B 0,C 180,E1 28875.496,E2 28875.496} C_VEL
LIN {X 0,Y 600.096,Z 636.79,A -85,B 0,C 180,E1 28874.242,E2 28874.242} C_VEL
LIN {X 0,Y 600.16,Z 620.933,A -85,B 0,C 180,E1 28873.1,E2 28873.1} C_VEL
LIN {X 0,Y 600.205,Z 603.942,A -85,B 0,C 180,E1 28872.101,E2 28872.101} C_VEL
LIN {X 0,Y 600.278,Z 586.855,A -85,B 0,C 180,E1 28871.295,E2 28871.295} C_VEL
LIN {X 0,Y 600.321,Z 568.317,A -85,B 0,C 180,E1 28870.622,E2 28870.622} C_VEL
LIN {X 0,Y 600.366,Z 549.69,A -85,B 0,C 180,E1 28870.136,E2 28870.136} C_VEL
LIN {X 0,Y 600.394,Z 529.98,A -85,B 0,C 180,E1 28869.813,E2 28869.813} C_VEL
LIN {X 0,Y 600.377,Z 334.753,A -85,B 0,C 180,E1 28867.35,E2 28867.35} C_VEL
LIN {X 0,Y 600.27,Z 329.595,A -85,B 0,C 180,E1 28866.957,E2 28866.957} C_VEL
LIN {X 0,Y 600.396,Z 292.735,A -85,B 0,C 180,E1 28863.813,E2 28863.813} C_VEL
LIN {X 0,Y 600.096,Z 288.551,A -85,B 0,C 180,E1 28863.431,E2 28863.431} C_VEL
LIN {X 0,Y 599.954,Z 287.79,A -85,B 0,C 180,E1 28863.259,E2 28863.259} C_VEL
LIN {X 0,Y 599.968,Z 287.751,A -85,B 0,C 180,E1 28860.065,E2 28860.065} C_VEL
LIN {X 0,Y 599.948,Z 287.747,A -85,B 0,C 180,E1 28856.865,E2 28856.865} C_VEL
LIN {X 0,Y 599.967,Z 287.753,A -85,B 0,C 180,E1 28853.604,E2 28853.604} C_VEL
LIN {X 0,Y 599.971,Z 287.744,A -85,B 0,C 180,E1 28850.338,E2 28850.338} C_VEL
LIN {X 0,Y 599.938,Z 287.748,A -85,B 0,C 180,E1 28847.16,E2 28847.16} C_VEL
LIN {X 0,Y 599.974,Z 287.747,A -85,B 0,C 180,E1 28844.022,E2 28844.022} C_VEL
LIN {X 0,Y 599.931,Z 287.749,A -85,B 0,C 180,E1 28840.919,E2 28840.919} C_VEL
LIN {X 0,Y 599.979,Z 287.753,A -85,B 0,C 180,E1 28837.706,E2 28837.706} C_VEL
LIN {X 0,Y 599.931,Z 287.748,A -85,B 0,C 180,E1 28834.585,E2 28834.585} C_VEL
LIN {X 0,Y 599.945,Z 287.752,A -85,B 0,C 180,E1 28831.331,E2 28831.331} C_VEL
LIN {X 0,Y 599.945,Z 287.748,A -85,B 0,C 180,E1 28828.25,E2 28828.25} C_VEL
LIN {X 0,Y 599.922,Z 287.751,A -85,B 0,C 180,E1 28825.045,E2 28825.045} C_VEL
LIN {X 0,Y 599.958,Z 287.749,A -85,B 0,C 180,E1 28822.023,E2 28822.023} C_VEL
LIN {X 0,Y 599.91,Z 287.752,A -85,B 0,C 180,E1 28818.865,E2 28818.865} C_VEL
LIN {X 0,Y 599.962,Z 287.75,A -85,B 0,C 180,E1 28815.862,E2 28815.862} C_VEL
LIN {X 0,Y 599.904,Z 287.752,A -85,B 0,C 180,E1 28812.807,E2 28812.807} C_VEL
LIN {X 0,Y 599.946,Z 287.751,A -85,B 0,C 180,E1 28809.884,E2 28809.884} C_VEL
LIN {X 0,Y 599.9,Z 287.753,A -85,B 0,C 180,E1 28806.796,E2 28806.796} C_VEL
LIN {X 0,Y 599.927,Z 287.753,A -85,B 0,C 180,E1 28803.918,E2 28803.918} C_VEL
LIN {X 0,Y 599.894,Z 287.754,A -85,B 0,C 180,E1 28800.764,E2 28800.764} C_VEL
LIN {X 0,Y 599.91,Z 287.753,A -85,B 0,C 180,E1 28797.994,E2 28797.994} C_VEL
LIN {X 0,Y 599.901,Z 287.753,A -85,B 0,C 180,E1 28794.741,E2 28794.741} C_VEL
LIN {X 0,Y 599.925,Z 287.753,A -85,B 0,C 180,E1 28791.856,E2 28791.856} C_VEL
LIN {X 0,Y 599.907,Z 287.752,A -85,B 0,C 180,E1 28788.658,E2 28788.658} C_VEL
LIN {X 0,Y 599.929,Z 287.752,A -85,B 0,C 180,E1 28785.819,E2 28785.819} C_VEL
LIN {X 0,Y 599.914,Z 287.751,A -85,B 0,C 180,E1 28782.643,E2 28782.643} C_VEL
LIN {X 0,Y 599.939,Z 287.753,A -85,B 0,C 180,E1 28779.717,E2 28779.717} C_VEL
LIN {X 0,Y 599.919,Z 287.75,A -85,B 0,C 180,E1 28776.526,E2 28776.526} C_VEL
LIN {X 0,Y 599.968,Z 287.754,A -85,B 0,C 180,E1 28773.473,E2 28773.473} C_VEL
LIN {X 0,Y 599.92,Z 287.75,A -85,B 0,C 180,E1 28770.331,E2 28770.331} C_VEL
LIN {X 0,Y 599.978,Z 287.751,A -85,B 0,C 180,E1 28767.207,E2 28767.207} C_VEL
LIN {X 0,Y 599.925,Z 287.748,A -85,B 0,C 180,E1 28764.08,E2 28764.08} C_VEL
LIN {X 0,Y 599.978,Z 287.747,A -85,B 0,C 180,E1 28760.947,E2 28760.947} C_VEL
LIN {X 0,Y 599.937,Z 287.748,A -85,B 0,C 180,E1 28757.806,E2 28757.806} C_VEL
LIN {X 0,Y 599.954,Z 287.745,A -85,B 0,C 180,E1 28754.497,E2 28754.497} C_VEL
LIN {X 0,Y 599.976,Z 287.753,A -85,B 0,C 180,E1 28751.272,E2 28751.272} C_VEL
LIN {X 0,Y 599.94,Z 287.749,A -85,B 0,C 180,E1 28748.07,E2 28748.07} C_VEL
LIN {X 0,Y 599.97,Z 287.745,A -85,B 0,C 180,E1 28744.923,E2 28744.923} C_VEL
LIN {X 0,Y 599.975,Z 287.98,A -85,B 0,C 180,E1 28743.91,E2 28743.91} C_VEL
LIN {X 0,Y 600.915,Z 290.689,A -85,B 0,C 180,E1 28743.646,E2 28743.646} C_VEL
LIN {X 0,Y 600.785,Z 342.119,A -85,B 0,C 180,E1 28740.725,E2 28740.725} C_VEL
LIN {X 0,Y 600.728,Z 391.1,A -85,B 0,C 180,E1 28738.048,E2 28738.048} C_VEL
LIN {X 0,Y 600.666,Z 596.888,A -85,B 0,C 180,E1 28735.353,E2 28735.353} C_VEL
LIN {X 0,Y 600.612,Z 654.257,A -85,B 0,C 180,E1 28734.583,E2 28734.583} C_VEL
LIN {X 0,Y 600.557,Z 674.736,A -85,B 0,C 180,E1 28734.124,E2 28734.124} C_VEL
LIN {X 0,Y 600.498,Z 693.797,A -85,B 0,C 180,E1 28733.527,E2 28733.527} C_VEL
LIN {X 0,Y 600.425,Z 713.624,A -85,B 0,C 180,E1 28732.726,E2 28732.726} C_VEL
LIN {X 0,Y 600.349,Z 732.065,A -85,B 0,C 180,E1 28731.801,E2 28731.801} C_VEL
LIN {X 0,Y 600.277,Z 750.54,A -85,B 0,C 180,E1 28730.678,E2 28730.678} C_VEL
LIN {X 0,Y 600.196,Z 768.576,A -85,B 0,C 180,E1 28729.36,E2 28729.36} C_VEL
LIN {X 0,Y 600.122,Z 785.371,A -85,B 0,C 180,E1 28727.902,E2 28727.902} C_VEL
LIN {X 0,Y 600.056,Z 800.903,A -85,B 0,C 180,E1 28726.307,E2 28726.307} C_VEL
LIN {X 0,Y 600.008,Z 814.366,A -85,B 0,C 180,E1 28724.672,E2 28724.672} C_VEL
LIN {X 0,Y 599.976,Z 826.017,A -85,B 0,C 180,E1 28723.001,E2 28723.001} C_VEL
LIN {X 0,Y 599.946,Z 836.327,A -85,B 0,C 180,E1 28721.244,E2 28721.244} C_VEL
LIN {X 0,Y 599.933,Z 845.34,A -85,B 0,C 180,E1 28719.378,E2 28719.378} C_VEL
LIN {X 0,Y 599.923,Z 852.38,A -85,B 0,C 180,E1 28717.566,E2 28717.566} C_VEL
LIN {X 0,Y 599.917,Z 858.002,A -85,B 0,C 180,E1 28715.643,E2 28715.643} C_VEL
LIN {X 0,Y 599.914,Z 861.924,A -85,B 0,C 180,E1 28713.727,E2 28713.727} C_VEL
LIN {X 0,Y 599.908,Z 864.306,A -85,B 0,C 180,E1 28711.719,E2 28711.719} C_VEL
LIN {X 0,Y 599.907,Z 864.962,A -85,B 0,C 180,E1 28709.809,E2 28709.809} C_VEL
LIN {X 0,Y 599.911,Z 864.039,A -85,B 0,C 180,E1 28707.899,E2 28707.899} C_VEL
LIN {X 0,Y 599.914,Z 861.451,A -85,B 0,C 180,E1 28705.986,E2 28705.986} C_VEL
LIN {X 0,Y 599.915,Z 857.242,A -85,B 0,C 180,E1 28704.069,E2 28704.069} C_VEL
LIN {X 0,Y 599.915,Z 851.327,A -85,B 0,C 180,E1 28702.145,E2 28702.145} C_VEL
LIN {X 0,Y 599.926,Z 844.017,A -85,B 0,C 180,E1 28700.31,E2 28700.31} C_VEL
LIN {X 0,Y 599.939,Z 834.772,A -85,B 0,C 180,E1 28698.464,E2 28698.464} C_VEL
LIN {X 0,Y 599.979,Z 824.098,A -85,B 0,C 180,E1 28696.705,E2 28696.705} C_VEL
LIN {X 0,Y 600.011,Z 812.04,A -85,B 0,C 180,E1 28695.032,E2 28695.032} C_VEL
LIN {X 0,Y 600.066,Z 798.599,A -85,B 0,C 180,E1 28693.446,E2 28693.446} C_VEL
LIN {X 0,Y 600.125,Z 783.715,A -85,B 0,C 180,E1 28691.948,E2 28691.948} C_VEL
LIN {X 0,Y 600.199,Z 767.851,A -85,B 0,C 180,E1 28690.584,E2 28690.584} C_VEL
LIN {X 0,Y 600.276,Z 750.539,A -85,B 0,C 180,E1 28689.322,E2 28689.322} C_VEL
LIN {X 0,Y 600.348,Z 732.063,A -85,B 0,C 180,E1 28688.199,E2 28688.199} C_VEL
LIN {X 0,Y 600.424,Z 713.621,A -85,B 0,C 180,E1 28687.274,E2 28687.274} C_VEL
LIN {X 0,Y 600.498,Z 693.796,A -85,B 0,C 180,E1 28686.473,E2 28686.473} C_VEL
LIN {X 0,Y 600.558,Z 674.063,A -85,B 0,C 180,E1 28685.859,E2 28685.859} C_VEL
LIN {X 0,Y 600.618,Z 653.731,A -85,B 0,C 180,E1 28685.407,E2 28685.407} C_VEL
LIN {X 0,Y 600.713,Z 509.726,A -85,B 0,C 180,E1 28683.515,E2 28683.515} C_VEL
LIN {X 0,Y 600.645,Z 390.371,A -85,B 0,C 180,E1 28681.932,E2 28681.932} C_VEL
LIN {X 0,Y 600.815,Z 334.206,A -85,B 0,C 180,E1 28678.832,E2 28678.832} C_VEL
LIN {X 0,Y 600.913,Z 290.688,A -85,B 0,C 180,E1 28676.354,E2 28676.354} C_VEL
LIN {X 0,Y 599.975,Z 287.98,A -85,B 0,C 180,E1 28676.09,E2 28676.09} C_VEL
LIN {X 0,Y 599.971,Z 287.749,A -85,B 0,C 180,E1 28673.016,E2 28673.016} C_VEL
LIN {X 0,Y 599.94,Z 287.747,A -85,B 0,C 180,E1 28669.838,E2 28669.838} C_VEL
LIN {X 0,Y 599.971,Z 287.751,A -85,B 0,C 180,E1 28666.602,E2 28666.602} C_VEL
LIN {X 0,Y 599.964,Z 287.746,A -85,B 0,C 180,E1 28663.362,E2 28663.362} C_VEL
LIN {X 0,Y 599.933,Z 287.751,A -85,B 0,C 180,E1 28660.097,E2 28660.097} C_VEL
LIN {X 0,Y 599.978,Z 287.747,A -85,B 0,C 180,E1 28656.985,E2 28656.985} C_VEL
LIN {X 0,Y 599.924,Z 287.75,A -85,B 0,C 180,E1 28653.825,E2 28653.825} C_VEL
LIN {X 0,Y 599.974,Z 287.753,A -85,B 0,C 180,E1 28650.66,E2 28650.66} C_VEL
LIN {X 0,Y 599.923,Z 287.749,A -85,B 0,C 180,E1 28647.547,E2 28647.547} C_VEL
LIN {X 0,Y 599.945,Z 287.752,A -85,B 0,C 180,E1 28644.308,E2 28644.308} C_VEL
LIN {X 0,Y 599.928,Z 287.75,A -85,B 0,C 180,E1 28641.304,E2 28641.304} C_VEL
LIN {X 0,Y 599.922,Z 287.752,A -85,B 0,C 180,E1 28638.059,E2 28638.059} C_VEL
LIN {X 0,Y 599.927,Z 287.751,A -85,B 0,C 180,E1 28635.168,E2 28635.168} C_VEL
LIN {X 0,Y 599.911,Z 287.753,A -85,B 0,C 180,E1 28631.927,E2 28631.927} C_VEL
LIN {X 0,Y 599.93,Z 287.751,A -85,B 0,C 180,E1 28629.013,E2 28629.013} C_VEL
LIN {X 0,Y 599.904,Z 287.753,A -85,B 0,C 180,E1 28625.835,E2 28625.835} C_VEL
LIN {X 0,Y 599.922,Z 287.752,A -85,B 0,C 180,E1 28622.961,E2 28622.961} C_VEL
LIN {X 0,Y 599.9,Z 287.754,A -85,B 0,C 180,E1 28619.809,E2 28619.809} C_VEL
LIN {X 0,Y 599.903,Z 287.753,A -85,B 0,C 180,E1 28617.038,E2 28617.038} C_VEL
LIN {X 0,Y 599.902,Z 287.753,A -85,B 0,C 180,E1 28613.78,E2 28613.78} C_VEL
LIN {X 0,Y 599.891,Z 287.754,A -85,B 0,C 180,E1 28613.462,E2 28613.462} C_VEL
LIN {X 0,Y 598.925,Z 287.88,A -85,B 0,C 180,E1 28612.726,E2 28612.726} C_VEL
LIN {X 0,Y 592.486,Z 288.687,A -85,B 0,C 180,E1 28610.608,E2 28610.608} C_VEL
LIN {X 0,Y 592.007,Z 288.741,A -85,B 0,C 180,E1 28610.125,E2 28610.125} C_VEL
LIN {X 0,Y 591.959,Z 288.742,A -85,B 0,C 180,E1 28607.216,E2 28607.216} C_VEL
LIN {X 0,Y 592.022,Z 288.74,A -85,B 0,C 180,E1 28604.121,E2 28604.121} C_VEL
LIN {X 0,Y 591.969,Z 288.741,A -85,B 0,C 180,E1 28601.077,E2 28601.077} C_VEL
LIN {X 0,Y 592.005,Z 288.739,A -85,B 0,C 180,E1 28597.874,E2 28597.874} C_VEL
LIN {X 0,Y 591.979,Z 288.739,A -85,B 0,C 180,E1 28594.916,E2 28594.916} C_VEL
LIN {X 0,Y 591.994,Z 288.738,A -85,B 0,C 180,E1 28591.633,E2 28591.633} C_VEL
LIN {X 0,Y 592,Z 288.741,A -85,B 0,C 180,E1 28588.654,E2 28588.654} C_VEL
LIN {X 0,Y 591.989,Z 288.738,A -85,B 0,C 180,E1 28585.424,E2 28585.424} C_VEL
LIN {X 0,Y 592.035,Z 288.742,A -85,B 0,C 180,E1 28582.312,E2 28582.312} C_VEL
LIN {X 0,Y 591.987,Z 288.738,A -85,B 0,C 180,E1 28579.169,E2 28579.169} C_VEL
LIN {X 0,Y 592.038,Z 288.737,A -85,B 0,C 180,E1 28576.007,E2 28576.007} C_VEL
LIN {X 0,Y 591.993,Z 288.736,A -85,B 0,C 180,E1 28572.86,E2 28572.86} C_VEL
LIN {X 0,Y 592.031,Z 288.733,A -85,B 0,C 180,E1 28569.635,E2 28569.635} C_VEL
LIN {X 0,Y 592.014,Z 288.741,A -85,B 0,C 180,E1 28566.476,E2 28566.476} C_VEL
LIN {X 0,Y 592.008,Z 288.736,A -85,B 0,C 180,E1 28563.175,E2 28563.175} C_VEL
LIN {X 0,Y 592.033,Z 288.742,A -85,B 0,C 180,E1 28559.959,E2 28559.959} C_VEL
LIN {X 0,Y 592.019,Z 288.846,A -85,B 0,C 180,E1 28556.907,E2 28556.907} C_VEL
LIN {X 0,Y 592.416,Z 290.475,A -85,B 0,C 180,E1 28556.675,E2 28556.675} C_VEL
LIN {X 0,Y 592.886,Z 293.544,A -85,B 0,C 180,E1 28556.382,E2 28556.382} C_VEL
LIN {X 0,Y 592.66,Z 329.764,A -85,B 0,C 180,E1 28553.251,E2 28553.251} C_VEL
LIN {X 0,Y 592.686,Z 334.316,A -85,B 0,C 180,E1 28552.882,E2 28552.882} C_VEL
LIN {X 0,Y 593.123,Z 338.906,A -85,B 0,C 180,E1 28552.792,E2 28552.792} C_VEL
LIN {X 0,Y 592.85,Z 542.359,A -85,B 0,C 180,E1 28550.181,E2 28550.181} C_VEL
LIN {X 0,Y 592.769,Z 561.326,A -85,B 0,C 180,E1 28549.752,E2 28549.752} C_VEL
LIN {X 0,Y 592.658,Z 579.704,A -85,B 0,C 180,E1 28549.15,E2 28549.15} C_VEL
LIN {X 0,Y 592.552,Z 597.183,A -85,B 0,C 180,E1 28548.393,E2 28548.393} C_VEL
LIN {X 0,Y 592.456,Z 613.883,A -85,B 0,C 180,E1 28547.481,E2 28547.481} C_VEL
LIN {X 0,Y 592.339,Z 629.714,A -85,B 0,C 180,E1 28546.423,E2 28546.423} C_VEL
LIN {X 0,Y 592.227,Z 644.624,A -85,B 0,C 180,E1 28545.22,E2 28545.22} C_VEL
LIN {X 0,Y 592.128,Z 658.532,A -85,B 0,C 180,E1 28543.873,E2 28543.873} C_VEL
LIN {X 0,Y 592.055,Z 671.336,A -85,B 0,C 180,E1 28542.384,E2 28542.384} C_VEL
LIN {X 0,Y 591.996,Z 682.577,A -85,B 0,C 180,E1 28540.805,E2 28540.805} C_VEL
LIN {X 0,Y 591.959,Z 692.273,A -85,B 0,C 180,E1 28539.135,E2 28539.135} C_VEL
LIN {X 0,Y 591.933,Z 700.036,A -85,B 0,C 180,E1 28537.463,E2 28537.463} C_VEL
LIN {X 0,Y 591.914,Z 706.272,A -85,B 0,C 180,E1 28535.72,E2 28535.72} C_VEL
LIN {X 0,Y 591.919,Z 710.78,A -85,B 0,C 180,E1 28533.971,E2 28533.971} C_VEL
LIN {X 0,Y 591.917,Z 713.737,A -85,B 0,C 180,E1 28532.13,E2 28532.13} C_VEL
LIN {X 0,Y 591.909,Z 714.929,A -85,B 0,C 180,E1 28530.29,E2 28530.29} C_VEL
LIN {X 0,Y 591.915,Z 714.38,A -85,B 0,C 180,E1 28528.451,E2 28528.451} C_VEL
LIN {X 0,Y 591.908,Z 712.08,A -85,B 0,C 180,E1 28526.611,E2 28526.611} C_VEL
LIN {X 0,Y 591.917,Z 708.215,A -85,B 0,C 180,E1 28524.864,E2 28524.864} C_VEL
LIN {X 0,Y 591.93,Z 702.632,A -85,B 0,C 180,E1 28523.112,E2 28523.112} C_VEL
LIN {X 0,Y 591.941,Z 695.636,A -85,B 0,C 180,E1 28521.452,E2 28521.452} C_VEL
LIN {X 0,Y 591.978,Z 686.777,A -85,B 0,C 180,E1 28519.785,E2 28519.785} C_VEL
LIN {X 0,Y 592.023,Z 676.47,A -85,B 0,C 180,E1 28518.209,E2 28518.209} C_VEL
LIN {X 0,Y 592.092,Z 664.733,A -85,B 0,C 180,E1 28516.723,E2 28516.723} C_VEL
LIN {X 0,Y 592.179,Z 651.547,A -85,B 0,C 180,E1 28515.33,E2 28515.33} C_VEL
LIN {X 0,Y 592.291,Z 636.779,A -85,B 0,C 180,E1 28514.029,E2 28514.029} C_VEL
LIN {X 0,Y 592.412,Z 620.92,A -85,B 0,C 180,E1 28512.872,E2 28512.872} C_VEL
LIN {X 0,Y 592.518,Z 603.836,A -85,B 0,C 180,E1 28511.856,E2 28511.856} C_VEL
LIN {X 0,Y 592.648,Z 586.494,A -85,B 0,C 180,E1 28511.031,E2 28511.031} C_VEL
LIN {X 0,Y 592.746,Z 568.083,A -85,B 0,C 180,E1 28510.358,E2 28510.358} C_VEL
LIN {X 0,Y 592.83,Z 549.495,A -85,B 0,C 180,E1 28509.87,E2 28509.87} C_VEL
LIN {X 0,Y 592.883,Z 529.801,A -85,B 0,C 180,E1 28509.545,E2 28509.545} C_VEL
LIN {X 0,Y 592.969,Z 335.979,A -85,B 0,C 180,E1 28507.074,E2 28507.074} C_VEL
LIN {X 0,Y 592.669,Z 334.111,A -85,B 0,C 180,E1 28507.017,E2 28507.017} C_VEL
LIN {X 0,Y 592.862,Z 297.641,A -85,B 0,C 180,E1 28503.886,E2 28503.886} C_VEL
LIN {X 0,Y 592.72,Z 291.498,A -85,B 0,C 180,E1 28503.34,E2 28503.34} C_VEL
LIN {X 0,Y 592.038,Z 288.941,A -85,B 0,C 180,E1 28503.041,E2 28503.041} C_VEL
LIN {X 0,Y 592.036,Z 288.74,A -85,B 0,C 180,E1 28499.848,E2 28499.848} C_VEL
LIN {X 0,Y 592.031,Z 288.734,A -85,B 0,C 180,E1 28496.543,E2 28496.543} C_VEL
LIN {X 0,Y 592.007,Z 288.74,A -85,B 0,C 180,E1 28493.283,E2 28493.283} C_VEL
LIN {X 0,Y 592.033,Z 288.735,A -85,B 0,C 180,E1 28490.063,E2 28490.063} C_VEL
LIN {X 0,Y 591.996,Z 288.735,A -85,B 0,C 180,E1 28486.975,E2 28486.975} C_VEL
LIN {X 0,Y 592.037,Z 288.739,A -85,B 0,C 180,E1 28483.823,E2 28483.823} C_VEL
LIN {X 0,Y 591.996,Z 288.737,A -85,B 0,C 180,E1 28480.684,E2 28480.684} C_VEL
LIN {X 0,Y 592.017,Z 288.742,A -85,B 0,C 180,E1 28477.446,E2 28477.446} C_VEL
LIN {X 0,Y 592.011,Z 288.736,A -85,B 0,C 180,E1 28474.325,E2 28474.325} C_VEL
LIN {X 0,Y 591.989,Z 288.74,A -85,B 0,C 180,E1 28471.098,E2 28471.098} C_VEL
LIN {X 0,Y 592.031,Z 288.736,A -85,B 0,C 180,E1 28468.002,E2 28468.002} C_VEL
LIN {X 0,Y 591.977,Z 288.738,A -85,B 0,C 180,E1 28464.871,E2 28464.871} C_VEL
LIN {X 0,Y 592.039,Z 288.74,A -85,B 0,C 180,E1 28461.746,E2 28461.746} C_VEL
LIN {X 0,Y 591.969,Z 288.74,A -85,B 0,C 180,E1 28458.644,E2 28458.644} C_VEL
LIN {X 0,Y 592.027,Z 288.741,A -85,B 0,C 180,E1 28455.477,E2 28455.477} C_VEL
LIN {X 0,Y 591.963,Z 288.741,A -85,B 0,C 180,E1 28452.486,E2 28452.486} C_VEL
LIN {X 0,Y 592.009,Z 288.74,A -85,B 0,C 180,E1 28449.331,E2 28449.331} C_VEL
LIN {X 0,Y 591.958,Z 288.742,A -85,B 0,C 180,E1 28446.401,E2 28446.401} C_VEL
LIN {X 0,Y 592.006,Z 288.741,A -85,B 0,C 180,E1 28443.292,E2 28443.292} C_VEL
LIN {X 0,Y 591.949,Z 288.743,A -85,B 0,C 180,E1 28440.387,E2 28440.387} C_VEL
LIN {X 0,Y 592.013,Z 288.741,A -85,B 0,C 180,E1 28437.29,E2 28437.29} C_VEL
LIN {X 0,Y 591.957,Z 288.742,A -85,B 0,C 180,E1 28434.281,E2 28434.281} C_VEL
LIN {X 0,Y 592.004,Z 288.74,A -85,B 0,C 180,E1 28431.115,E2 28431.115} C_VEL
LIN {X 0,Y 591.964,Z 288.742,A -85,B 0,C 180,E1 28428.207,E2 28428.207} C_VEL
LIN {X 0,Y 592.008,Z 288.74,A -85,B 0,C 180,E1 28425.025,E2 28425.025} C_VEL
LIN {X 0,Y 591.972,Z 288.741,A -85,B 0,C 180,E1 28422.097,E2 28422.097} C_VEL
LIN {X 0,Y 592.009,Z 288.738,A -85,B 0,C 180,E1 28418.916,E2 28418.916} C_VEL
LIN {X 0,Y 591.981,Z 288.74,A -85,B 0,C 180,E1 28415.981,E2 28415.981} C_VEL
LIN {X 0,Y 591.995,Z 288.737,A -85,B 0,C 180,E1 28412.652,E2 28412.652} C_VEL
LIN {X 0,Y 592.017,Z 288.742,A -85,B 0,C 180,E1 28409.558,E2 28409.558} C_VEL
LIN {X 0,Y 591.988,Z 288.738,A -85,B 0,C 180,E1 28406.359,E2 28406.359} C_VEL
LIN {X 0,Y 592.039,Z 288.738,A -85,B 0,C 180,E1 28403.284,E2 28403.284} C_VEL
LIN {X 0,Y 591.99,Z 288.739,A -85,B 0,C 180,E1 28400.065,E2 28400.065} C_VEL
LIN {X 0,Y 592.037,Z 288.737,A -85,B 0,C 180,E1 28396.977,E2 28396.977} C_VEL
LIN {X 0,Y 591.999,Z 288.738,A -85,B 0,C 180,E1 28393.824,E2 28393.824} C_VEL
LIN {X 0,Y 592.026,Z 288.732,A -85,B 0,C 180,E1 28390.537,E2 28390.537} C_VEL
LIN {X 0,Y 592.029,Z 288.739,A -85,B 0,C 180,E1 28387.302,E2 28387.302} C_VEL
LIN {X 0,Y 592.054,Z 288.974,A -85,B 0,C 180,E1 28384.365,E2 28384.365} C_VEL
LIN {X 0,Y 593.469,Z 292.667,A -85,B 0,C 180,E1 28384.009,E2 28384.009} C_VEL
LIN {X 0,Y 593.995,Z 294.645,A -85,B 0,C 180,E1 28383.859,E2 28383.859} C_VEL
LIN {X 0,Y 593.635,Z 348.076,A -85,B 0,C 180,E1 28380.797,E2 28380.797} C_VEL
LIN {X 0,Y 593.492,Z 391.113,A -85,B 0,C 180,E1 28378.421,E2 28378.421} C_VEL
LIN {X 0,Y 593.697,Z 408.263,A -85,B 0,C 180,E1 28378.179,E2 28378.179} C_VEL
LIN {X 0,Y 593.337,Z 653.628,A -85,B 0,C 180,E1 28374.917,E2 28374.917} C_VEL
LIN {X 0,Y 593.228,Z 673.971,A -85,B 0,C 180,E1 28374.461,E2 28374.461} C_VEL
LIN {X 0,Y 593.104,Z 693.8,A -85,B 0,C 180,E1 28373.838,E2 28373.838} C_VEL
LIN {X 0,Y 592.951,Z 713.627,A -85,B 0,C 180,E1 28373.029,E2 28373.029} C_VEL
LIN {X 0,Y 592.804,Z 732.062,A -85,B 0,C 180,E1 28372.093,E2 28372.093} C_VEL
LIN {X 0,Y 592.653,Z 750.537,A -85,B 0,C 180,E1 28370.956,E2 28370.956} C_VEL
LIN {X 0,Y 592.491,Z 768.577,A -85,B 0,C 180,E1 28369.622,E2 28369.622} C_VEL
LIN {X 0,Y 592.337,Z 785.5,A -85,B 0,C 180,E1 28368.133,E2 28368.133} C_VEL
LIN {X 0,Y 592.214,Z 800.453,A -85,B 0,C 180,E1 28366.578,E2 28366.578} C_VEL
LIN {X 0,Y 592.109,Z 813.592,A -85,B 0,C 180,E1 28364.972,E2 28364.972} C_VEL
LIN {X 0,Y 592.04,Z 825.379,A -85,B 0,C 180,E1 28363.278,E2 28363.278} C_VEL
LIN {X 0,Y 591.978,Z 836.328,A -85,B 0,C 180,E1 28361.397,E2 28361.397} C_VEL
LIN {X 0,Y 591.945,Z 845.249,A -85,B 0,C 180,E1 28359.528,E2 28359.528} C_VEL
LIN {X 0,Y 591.931,Z 852.38,A -85,B 0,C 180,E1 28357.668,E2 28357.668} C_VEL
LIN {X 0,Y 591.918,Z 858.002,A -85,B 0,C 180,E1 28355.72,E2 28355.72} C_VEL
LIN {X 0,Y 591.915,Z 861.925,A -85,B 0,C 180,E1 28353.777,E2 28353.777} C_VEL
LIN {X 0,Y 591.908,Z 864.307,A -85,B 0,C 180,E1 28351.742,E2 28351.742} C_VEL
LIN {X 0,Y 591.907,Z 864.962,A -85,B 0,C 180,E1 28349.806,E2 28349.806} C_VEL
LIN {X 0,Y 591.91,Z 864.038,A -85,B 0,C 180,E1 28347.87,E2 28347.87} C_VEL
LIN {X 0,Y 591.913,Z 861.451,A -85,B 0,C 180,E1 28345.932,E2 28345.932} C_VEL
LIN {X 0,Y 591.921,Z 857.243,A -85,B 0,C 180,E1 28343.989,E2 28343.989} C_VEL
LIN {X 0,Y 591.922,Z 851.328,A -85,B 0,C 180,E1 28342.038,E2 28342.038} C_VEL
LIN {X 0,Y 591.944,Z 844.017,A -85,B 0,C 180,E1 28340.178,E2 28340.178} C_VEL
LIN {X 0,Y 591.977,Z 834.773,A -85,B 0,C 180,E1 28338.306,E2 28338.306} C_VEL
LIN {X 0,Y 592.042,Z 824.099,A -85,B 0,C 180,E1 28336.523,E2 28336.523} C_VEL
LIN {X 0,Y 592.12,Z 812.041,A -85,B 0,C 180,E1 28334.827,E2 28334.827} C_VEL
LIN {X 0,Y 592.221,Z 798.333,A -85,B 0,C 180,E1 28333.191,E2 28333.191} C_VEL
LIN {X 0,Y 592.345,Z 783.715,A -85,B 0,C 180,E1 28331.702,E2 28331.702} C_VEL
LIN {X 0,Y 592.498,Z 767.944,A -85,B 0,C 180,E1 28330.329,E2 28330.329} C_VEL
LIN {X 0,Y 592.653,Z 750.536,A -85,B 0,C 180,E1 28329.044,E2 28329.044} C_VEL
LIN {X 0,Y 592.804,Z 732.06,A -85,B 0,C 180,E1 28327.907,E2 28327.907} C_VEL
LIN {X 0,Y 592.951,Z 713.624,A -85,B 0,C 180,E1 28326.971,E2 28326.971} C_VEL
LIN {X 0,Y 593.104,Z 693.798,A -85,B 0,C 180,E1 28326.161,E2 28326.161} C_VEL
LIN {X 0,Y 593.228,Z 673.972,A -85,B 0,C 180,E1 28325.539,E2 28325.539} C_VEL
LIN {X 0,Y 593.337,Z 653.731,A -85,B 0,C 180,E1 28325.085,E2 28325.085} C_VEL
LIN {X 0,Y 593.585,Z 495.247,A -85,B 0,C 180,E1 28322.979,E2 28322.979} C_VEL
LIN {X 0,Y 593.535,Z 391.421,A -85,B 0,C 180,E1 28321.586,E2 28321.586} C_VEL
LIN {X 0,Y 593.423,Z 386.627,A -85,B 0,C 180,E1 28321.358,E2 28321.358} C_VEL
LIN {X 0,Y 593.764,Z 330.25,A -85,B 0,C 180,E1 28318.193,E2 28318.193} C_VEL
LIN {X 0,Y 593.912,Z 293.959,A -85,B 0,C 180,E1 28316.096,E2 28316.096} C_VEL
LIN {X 0,Y 592.08,Z 289.145,A -85,B 0,C 180,E1 28315.666,E2 28315.666} C_VEL
LIN {X 0,Y 592.035,Z 288.729,A -85,B 0,C 180,E1 28315.311,E2 28315.311} C_VEL
LIN {X 0,Y 592.003,Z 288.741,A -85,B 0,C 180,E1 28312.188,E2 28312.188} C_VEL
LIN {X 0,Y 592.032,Z 288.736,A -85,B 0,C 180,E1 28309.018,E2 28309.018} C_VEL
LIN {X 0,Y 591.997,Z 288.736,A -85,B 0,C 180,E1 28305.873,E2 28305.873} C_VEL
LIN {X 0,Y 592.033,Z 288.74,A -85,B 0,C 180,E1 28302.724,E2 28302.724} C_VEL
LIN {X 0,Y 592.002,Z 288.737,A -85,B 0,C 180,E1 28299.548,E2 28299.548} C_VEL
LIN {X 0,Y 591.998,Z 288.737,A -85,B 0,C 180,E1 28296.237,E2 28296.237} C_VEL
LIN {X 0,Y 592.03,Z 288.736,A -85,B 0,C 180,E1 28293.107,E2 28293.107} C_VEL
LIN {X 0,Y 591.982,Z 288.74,A -85,B 0,C 180,E1 28289.884,E2 28289.884} C_VEL
LIN {X 0,Y 592.038,Z 288.738,A -85,B 0,C 180,E1 28286.803,E2 28286.803} C_VEL
LIN {X 0,Y 591.976,Z 288.739,A -85,B 0,C 180,E1 28283.702,E2 28283.702} C_VEL
LIN {X 0,Y 592.033,Z 288.744,A -85,B 0,C 180,E1 28280.566,E2 28280.566} C_VEL
LIN {X 0,Y 591.971,Z 288.74,A -85,B 0,C 180,E1 28277.496,E2 28277.496} C_VEL
LIN {X 0,Y 592.017,Z 288.74,A -85,B 0,C 180,E1 28274.375,E2 28274.375} C_VEL
LIN {X 0,Y 591.967,Z 288.741,A -85,B 0,C 180,E1 28271.398,E2 28271.398} C_VEL
LIN {X 0,Y 591.992,Z 288.741,A -85,B 0,C 180,E1 28268.156,E2 28268.156} C_VEL
LIN {X 0,Y 591.966,Z 288.742,A -85,B 0,C 180,E1 28265.233,E2 28265.233} C_VEL
LIN {X 0,Y 591.971,Z 288.742,A -85,B 0,C 180,E1 28261.936,E2 28261.936} C_VEL
LIN {X 0,Y 591.961,Z 288.743,A -85,B 0,C 180,E1 28259.129,E2 28259.129} C_VEL
LIN {X 0,Y 591.964,Z 288.742,A -85,B 0,C 180,E1 28255.835,E2 28255.835} C_VEL
LIN {X 0,Y 591.967,Z 288.743,A -85,B 0,C 180,E1 28253.015,E2 28253.015} C_VEL
LIN {X 0,Y 592.007,Z 288.741,A -85,B 0,C 180,E1 28250.125,E2 28250.125} C_VEL
LIN {X 0,Y 590.944,Z 288.872,A -85,B 0,C 180,E1 28249.379,E2 28249.379} C_VEL
LIN {X 0,Y 584.531,Z 289.669,A -85,B 0,C 180,E1 28247.288,E2 28247.288} C_VEL
LIN {X 0,Y 584.053,Z 289.731,A -85,B 0,C 180,E1 28246.743,E2 28246.743} C_VEL
LIN {X 0,Y 584.028,Z 289.73,A -85,B 0,C 180,E1 28243.489,E2 28243.489} C_VEL
LIN {X 0,Y 584.093,Z 289.729,A -85,B 0,C 180,E1 28240.396,E2 28240.396} C_VEL
LIN {X 0,Y 584.03,Z 289.73,A -85,B 0,C 180,E1 28237.237,E2 28237.237} C_VEL
LIN {X 0,Y 584.096,Z 289.728,A -85,B 0,C 180,E1 28234.118,E2 28234.118} C_VEL
LIN {X 0,Y 584.039,Z 289.729,A -85,B 0,C 180,E1 28231.02,E2 28231.02} C_VEL
LIN {X 0,Y 584.083,Z 289.726,A -85,B 0,C 180,E1 28227.833,E2 28227.833} C_VEL
LIN {X 0,Y 584.054,Z 289.73,A -85,B 0,C 180,E1 28224.743,E2 28224.743} C_VEL
LIN {X 0,Y 584.059,Z 289.726,A -85,B 0,C 180,E1 28221.454,E2 28221.454} C_VEL
LIN {X 0,Y 584.097,Z 289.73,A -85,B 0,C 180,E1 28218.249,E2 28218.249} C_VEL
LIN {X 0,Y 584.052,Z 289.726,A -85,B 0,C 180,E1 28215.006,E2 28215.006} C_VEL
LIN {X 0,Y 584.096,Z 289.727,A -85,B 0,C 180,E1 28211.872,E2 28211.872} C_VEL
LIN {X 0,Y 584.062,Z 289.727,A -85,B 0,C 180,E1 28208.669,E2 28208.669} C_VEL
LIN {X 0,Y 584.078,Z 289.723,A -85,B 0,C 180,E1 28205.352,E2 28205.352} C_VEL
LIN {X 0,Y 584.097,Z 289.728,A -85,B 0,C 180,E1 28202.076,E2 28202.076} C_VEL
LIN {X 0,Y 584.065,Z 289.73,A -85,B 0,C 180,E1 28198.865,E2 28198.865} C_VEL
LIN {X 0,Y 584.11,Z 289.95,A -85,B 0,C 180,E1 28197.196,E2 28197.196} C_VEL
LIN {X 0,Y 585.382,Z 295.394,A -85,B 0,C 180,E1 28196.583,E2 28196.583} C_VEL
LIN {X 0,Y 585.044,Z 331.749,A -85,B 0,C 180,E1 28193.4,E2 28193.4} C_VEL
LIN {X 0,Y 585.16,Z 334.92,A -85,B 0,C 180,E1 28193.179,E2 28193.179} C_VEL
LIN {X 0,Y 585.746,Z 339.839,A -85,B 0,C 180,E1 28193.084,E2 28193.084} C_VEL
LIN {X 0,Y 585.337,Z 542.393,A -85,B 0,C 180,E1 28190.452,E2 28190.452} C_VEL
LIN {X 0,Y 585.221,Z 561.393,A -85,B 0,C 180,E1 28190.016,E2 28190.016} C_VEL
LIN {X 0,Y 585.062,Z 579.718,A -85,B 0,C 180,E1 28189.409,E2 28189.409} C_VEL
LIN {X 0,Y 584.902,Z 597.193,A -85,B 0,C 180,E1 28188.642,E2 28188.642} C_VEL
LIN {X 0,Y 584.745,Z 613.89,A -85,B 0,C 180,E1 28187.719,E2 28187.719} C_VEL
LIN {X 0,Y 584.568,Z 629.719,A -85,B 0,C 180,E1 28186.648,E2 28186.648} C_VEL
LIN {X 0,Y 584.401,Z 644.602,A -85,B 0,C 180,E1 28185.431,E2 28185.431} C_VEL
LIN {X 0,Y 584.248,Z 658.538,A -85,B 0,C 180,E1 28184.064,E2 28184.064} C_VEL
LIN {X 0,Y 584.131,Z 671.343,A -85,B 0,C 180,E1 28182.555,E2 28182.555} C_VEL
LIN {X 0,Y 584.043,Z 682.582,A -85,B 0,C 180,E1 28180.954,E2 28180.954} C_VEL
LIN {X 0,Y 583.984,Z 692.278,A -85,B 0,C 180,E1 28179.261,E2 28179.261} C_VEL
LIN {X 0,Y 583.945,Z 700.219,A -85,B 0,C 180,E1 28177.521,E2 28177.521} C_VEL
LIN {X 0,Y 583.917,Z 706.275,A -85,B 0,C 180,E1 28175.798,E2 28175.798} C_VEL
LIN {X 0,Y 583.919,Z 710.782,A -85,B 0,C 180,E1 28174.026,E2 28174.026} C_VEL
LIN {X 0,Y 583.916,Z 713.739,A -85,B 0,C 180,E1 28172.159,E2 28172.159} C_VEL
LIN {X 0,Y 583.909,Z 714.929,A -85,B 0,C 180,E1 28170.294,E2 28170.294} C_VEL
LIN {X 0,Y 583.914,Z 714.38,A -85,B 0,C 180,E1 28168.43,E2 28168.43} C_VEL
LIN {X 0,Y 583.908,Z 712.079,A -85,B 0,C 180,E1 28166.564,E2 28166.564} C_VEL
LIN {X 0,Y 583.919,Z 708.214,A -85,B 0,C 180,E1 28164.793,E2 28164.793} C_VEL
LIN {X 0,Y 583.938,Z 702.63,A -85,B 0,C 180,E1 28163.017,E2 28163.017} C_VEL
LIN {X 0,Y 583.956,Z 695.634,A -85,B 0,C 180,E1 28161.334,E2 28161.334} C_VEL
LIN {X 0,Y 584.014,Z 686.774,A -85,B 0,C 180,E1 28159.644,E2 28159.644} C_VEL
LIN {X 0,Y 584.083,Z 676.467,A -85,B 0,C 180,E1 28158.046,E2 28158.046} C_VEL
LIN {X 0,Y 584.19,Z 664.728,A -85,B 0,C 180,E1 28156.54,E2 28156.54} C_VEL
LIN {X 0,Y 584.326,Z 651.539,A -85,B 0,C 180,E1 28155.128,E2 28155.128} C_VEL
LIN {X 0,Y 584.491,Z 636.768,A -85,B 0,C 180,E1 28153.81,E2 28153.81} C_VEL
LIN {X 0,Y 584.673,Z 620.906,A -85,B 0,C 180,E1 28152.638,E2 28152.638} C_VEL
LIN {X 0,Y 584.841,Z 603.926,A -85,B 0,C 180,E1 28151.614,E2 28151.614} C_VEL
LIN {X 0,Y 585.026,Z 586.92,A -85,B 0,C 180,E1 28150.793,E2 28150.793} C_VEL
LIN {X 0,Y 585.179,Z 568.39,A -85,B 0,C 180,E1 28150.103,E2 28150.103} C_VEL
LIN {X 0,Y 585.306,Z 549.625,A -85,B 0,C 180,E1 28149.603,E2 28149.603} C_VEL
LIN {X 0,Y 585.385,Z 529.877,A -85,B 0,C 180,E1 28149.272,E2 28149.272} C_VEL
LIN {X 0,Y 585.591,Z 337.201,A -85,B 0,C 180,E1 28146.785,E2 28146.785} C_VEL
LIN {X 0,Y 585.049,Z 334.004,A -85,B 0,C 180,E1 28146.695,E2 28146.695} C_VEL
LIN {X 0,Y 585.363,Z 297.512,A -85,B 0,C 180,E1 28143.515,E2 28143.515} C_VEL
LIN {X 0,Y 585.222,Z 293.947,A -85,B 0,C 180,E1 28143.19,E2 28143.19} C_VEL
LIN {X 0,Y 584.111,Z 289.888,A -85,B 0,C 180,E1 28142.694,E2 28142.694} C_VEL
LIN {X 0,Y 584.073,Z 289.725,A -85,B 0,C 180,E1 28139.328,E2 28139.328} C_VEL
LIN {X 0,Y 584.092,Z 289.727,A -85,B 0,C 180,E1 28136.08,E2 28136.08} C_VEL
LIN {X 0,Y 584.064,Z 289.726,A -85,B 0,C 180,E1 28132.916,E2 28132.916} C_VEL
LIN {X 0,Y 584.094,Z 289.732,A -85,B 0,C 180,E1 28129.62,E2 28129.62} C_VEL
LIN {X 0,Y 584.089,Z 289.719,A -85,B 0,C 180,E1 28126.382,E2 28126.382} C_VEL
LIN {X 0,Y 584.061,Z 289.729,A -85,B 0,C 180,E1 28123.176,E2 28123.176} C_VEL
LIN {X 0,Y 584.098,Z 289.725,A -85,B 0,C 180,E1 28120.064,E2 28120.064} C_VEL
LIN {X 0,Y 584.05,Z 289.728,A -85,B 0,C 180,E1 28116.922,E2 28116.922} C_VEL
LIN {X 0,Y 584.099,Z 289.729,A -85,B 0,C 180,E1 28113.705,E2 28113.705} C_VEL
LIN {X 0,Y 584.05,Z 289.727,A -85,B 0,C 180,E1 28110.561,E2 28110.561} C_VEL
LIN {X 0,Y 584.065,Z 289.731,A -85,B 0,C 180,E1 28107.309,E2 28107.309} C_VEL
LIN {X 0,Y 584.059,Z 289.725,A -85,B 0,C 180,E1 28104.259,E2 28104.259} C_VEL
LIN {X 0,Y 584.04,Z 289.729,A -85,B 0,C 180,E1 28100.965,E2 28100.965} C_VEL
LIN {X 0,Y 584.091,Z 289.727,A -85,B 0,C 180,E1 28097.844,E2 28097.844} C_VEL
LIN {X 0,Y 584.027,Z 289.727,A -85,B 0,C 180,E1 28094.678,E2 28094.678} C_VEL
LIN {X 0,Y 584.096,Z 289.732,A -85,B 0,C 180,E1 28091.554,E2 28091.554} C_VEL
LIN {X 0,Y 584.021,Z 289.727,A -85,B 0,C 180,E1 28088.467,E2 28088.467} C_VEL
LIN {X 0,Y 584.068,Z 289.731,A -85,B 0,C 180,E1 28085.304,E2 28085.304} C_VEL
LIN {X 0,Y 584.015,Z 289.729,A -85,B 0,C 180,E1 28082.355,E2 28082.355} C_VEL
LIN {X 0,Y 584.058,Z 289.731,A -85,B 0,C 180,E1 28079.215,E2 28079.215} C_VEL
LIN {X 0,Y 584.016,Z 289.73,A -85,B 0,C 180,E1 28076.27,E2 28076.27} C_VEL
LIN {X 0,Y 584.06,Z 289.729,A -85,B 0,C 180,E1 28073.118,E2 28073.118} C_VEL
LIN {X 0,Y 584.026,Z 289.73,A -85,B 0,C 180,E1 28070.143,E2 28070.143} C_VEL
LIN {X 0,Y 584.045,Z 289.726,A -85,B 0,C 180,E1 28066.839,E2 28066.839} C_VEL
LIN {X 0,Y 584.045,Z 289.731,A -85,B 0,C 180,E1 28063.899,E2 28063.899} C_VEL
LIN {X 0,Y 584.04,Z 289.728,A -85,B 0,C 180,E1 28060.603,E2 28060.603} C_VEL
LIN {X 0,Y 584.08,Z 289.731,A -85,B 0,C 180,E1 28057.559,E2 28057.559} C_VEL
LIN {X 0,Y 584.038,Z 289.729,A -85,B 0,C 180,E1 28054.334,E2 28054.334} C_VEL
LIN {X 0,Y 584.102,Z 289.729,A -85,B 0,C 180,E1 28051.212,E2 28051.212} C_VEL
LIN {X 0,Y 584.045,Z 289.728,A -85,B 0,C 180,E1 28048.063,E2 28048.063} C_VEL
LIN {X 0,Y 584.094,Z 289.719,A -85,B 0,C 180,E1 28044.889,E2 28044.889} C_VEL
LIN {X 0,Y 584.064,Z 289.729,A -85,B 0,C 180,E1 28041.705,E2 28041.705} C_VEL
LIN {X 0,Y 584.061,Z 289.719,A -85,B 0,C 180,E1 28038.378,E2 28038.378} C_VEL
LIN {X 0,Y 584.099,Z 289.729,A -85,B 0,C 180,E1 28035.265,E2 28035.265} C_VEL
LIN {X 0,Y 584.058,Z 289.728,A -85,B 0,C 180,E1 28032.015,E2 28032.015} C_VEL
LIN {X 0,Y 584.096,Z 289.728,A -85,B 0,C 180,E1 28028.843,E2 28028.843} C_VEL
LIN {X 0,Y 584.075,Z 289.734,A -85,B 0,C 180,E1 28025.593,E2 28025.593} C_VEL
LIN {X 0,Y 584.139,Z 290.034,A -85,B 0,C 180,E1 28024.823,E2 28024.823} C_VEL
LIN {X 0,Y 587.056,Z 297.689,A -85,B 0,C 180,E1 28024.133,E2 28024.133} C_VEL
LIN {X 0,Y 586.515,Z 351.021,A -85,B 0,C 180,E1 28021.042,E2 28021.042} C_VEL
LIN {X 0,Y 586.276,Z 391.086,A -85,B 0,C 180,E1 28018.804,E2 28018.804} C_VEL
LIN {X 0,Y 586.677,Z 397.066,A -85,B 0,C 180,E1 28018.7,E2 28018.7} C_VEL
LIN {X 0,Y 586.142,Z 631.431,A -85,B 0,C 180,E1 28015.567,E2 28015.567} C_VEL
LIN {X 0,Y 586.031,Z 658.151,A -85,B 0,C 180,E1 28015.156,E2 28015.156} C_VEL
LIN {X 0,Y 585.863,Z 678.255,A -85,B 0,C 180,E1 28014.669,E2 28014.669} C_VEL
LIN {X 0,Y 585.699,Z 698.068,A -85,B 0,C 180,E1 28014.003,E2 28014.003} C_VEL
LIN {X 0,Y 585.469,Z 716.988,A -85,B 0,C 180,E1 28013.181,E2 28013.181} C_VEL
LIN {X 0,Y 585.221,Z 735.717,A -85,B 0,C 180,E1 28012.178,E2 28012.178} C_VEL
LIN {X 0,Y 584.966,Z 754.196,A -85,B 0,C 180,E1 28010.982,E2 28010.982} C_VEL
LIN {X 0,Y 584.73,Z 771.625,A -85,B 0,C 180,E1 28009.633,E2 28009.633} C_VEL
LIN {X 0,Y 584.524,Z 787.62,A -85,B 0,C 180,E1 28008.17,E2 28008.17} C_VEL
LIN {X 0,Y 584.348,Z 802.207,A -85,B 0,C 180,E1 28006.603,E2 28006.603} C_VEL
LIN {X 0,Y 584.197,Z 815.861,A -85,B 0,C 180,E1 28004.875,E2 28004.875} C_VEL
LIN {X 0,Y 584.091,Z 827.93,A -85,B 0,C 180,E1 28003.059,E2 28003.059} C_VEL
LIN {X 0,Y 584.005,Z 838.399,A -85,B 0,C 180,E1 28001.155,E2 28001.155} C_VEL
LIN {X 0,Y 583.962,Z 846.875,A -85,B 0,C 180,E1 27999.262,E2 27999.262} C_VEL
LIN {X 0,Y 583.93,Z 853.9,A -85,B 0,C 180,E1 27997.279,E2 27997.279} C_VEL
LIN {X 0,Y 583.914,Z 859.144,A -85,B 0,C 180,E1 27995.305,E2 27995.305} C_VEL
LIN {X 0,Y 583.909,Z 862.71,A -85,B 0,C 180,E1 27993.338,E2 27993.338} C_VEL
LIN {X 0,Y 583.905,Z 864.639,A -85,B 0,C 180,E1 27991.275,E2 27991.275} C_VEL
LIN {X 0,Y 583.904,Z 864.851,A -85,B 0,C 180,E1 27989.313,E2 27989.313} C_VEL
LIN {X 0,Y 583.91,Z 863.392,A -85,B 0,C 180,E1 27987.252,E2 27987.252} C_VEL
LIN {X 0,Y 583.918,Z 860.169,A -85,B 0,C 180,E1 27985.187,E2 27985.187} C_VEL
LIN {X 0,Y 583.931,Z 855.414,A -85,B 0,C 180,E1 27983.215,E2 27983.215} C_VEL
LIN {X 0,Y 583.948,Z 848.851,A -85,B 0,C 180,E1 27981.235,E2 27981.235} C_VEL
LIN {X 0,Y 583.98,Z 840.795,A -85,B 0,C 180,E1 27979.344,E2 27979.344} C_VEL
LIN {X 0,Y 584.05,Z 830.838,A -85,B 0,C 180,E1 27977.443,E2 27977.443} C_VEL
LIN {X 0,Y 584.159,Z 819.391,A -85,B 0,C 180,E1 27975.63,E2 27975.63} C_VEL
LIN {X 0,Y 584.299,Z 806.451,A -85,B 0,C 180,E1 27973.906,E2 27973.906} C_VEL
LIN {X 0,Y 584.476,Z 791.978,A -85,B 0,C 180,E1 27972.272,E2 27972.272} C_VEL
LIN {X 0,Y 584.683,Z 776.45,A -85,B 0,C 180,E1 27970.781,E2 27970.781} C_VEL
LIN {X 0,Y 584.922,Z 759.28,A -85,B 0,C 180,E1 27969.383,E2 27969.383} C_VEL
LIN {X 0,Y 585.174,Z 740.916,A -85,B 0,C 180,E1 27968.132,E2 27968.132} C_VEL
LIN {X 0,Y 585.388,Z 722.299,A -85,B 0,C 180,E1 27967.082,E2 27967.082} C_VEL
LIN {X 0,Y 585.612,Z 702.731,A -85,B 0,C 180,E1 27966.185,E2 27966.185} C_VEL
LIN {X 0,Y 585.833,Z 682.304,A -85,B 0,C 180,E1 27965.456,E2 27965.456} C_VEL
LIN {X 0,Y 586.013,Z 662.109,A -85,B 0,C 180,E1 27964.925,E2 27964.925} C_VEL
LIN {X 0,Y 586.122,Z 641.479,A -85,B 0,C 180,E1 27964.566,E2 27964.566} C_VEL
LIN {X 0,Y 586.657,Z 403.425,A -85,B 0,C 180,E1 27961.386,E2 27961.386} C_VEL
LIN {X 0,Y 586.434,Z 392.169,A -85,B 0,C 180,E1 27961.22,E2 27961.22} C_VEL
LIN {X 0,Y 586.183,Z 389.594,A -85,B 0,C 180,E1 27961.138,E2 27961.138} C_VEL
LIN {X 0,Y 586.704,Z 333.118,A -85,B 0,C 180,E1 27957.932,E2 27957.932} C_VEL
LIN {X 0,Y 586.959,Z 297.044,A -85,B 0,C 180,E1 27955.822,E2 27955.822} C_VEL
LIN {X 0,Y 584.146,Z 290.078,A -85,B 0,C 180,E1 27955.182,E2 27955.182} C_VEL
LIN {X 0,Y 584.087,Z 289.73,A -85,B 0,C 180,E1 27954.57,E2 27954.57} C_VEL
LIN {X 0,Y 584.096,Z 289.726,A -85,B 0,C 180,E1 27951.314,E2 27951.314} C_VEL
LIN {X 0,Y 584.061,Z 289.729,A -85,B 0,C 180,E1 27948.116,E2 27948.116} C_VEL
LIN {X 0,Y 584.097,Z 289.726,A -85,B 0,C 180,E1 27944.874,E2 27944.874} C_VEL
LIN {X 0,Y 584.057,Z 289.719,A -85,B 0,C 180,E1 27941.723,E2 27941.723} C_VEL
LIN {X 0,Y 584.077,Z 289.729,A -85,B 0,C 180,E1 27938.419,E2 27938.419} C_VEL
LIN {X 0,Y 584.083,Z 289.719,A -85,B 0,C 180,E1 27935.232,E2 27935.232} C_VEL
LIN {X 0,Y 584.05,Z 289.729,A -85,B 0,C 180,E1 27932.053,E2 27932.053} C_VEL
LIN {X 0,Y 584.098,Z 289.728,A -85,B 0,C 180,E1 27928.863,E2 27928.863} C_VEL
LIN {X 0,Y 584.039,Z 289.729,A -85,B 0,C 180,E1 27925.775,E2 27925.775} C_VEL
LIN {X 0,Y 584.102,Z 289.728,A -85,B 0,C 180,E1 27922.653,E2 27922.653} C_VEL
LIN {X 0,Y 584.037,Z 289.728,A -85,B 0,C 180,E1 27919.502,E2 27919.502} C_VEL
LIN {X 0,Y 584.069,Z 289.731,A -85,B 0,C 180,E1 27916.305,E2 27916.305} C_VEL
LIN {X 0,Y 584.033,Z 289.726,A -85,B 0,C 180,E1 27913.363,E2 27913.363} C_VEL
LIN {X 0,Y 584.043,Z 289.73,A -85,B 0,C 180,E1 27910.056,E2 27910.056} C_VEL
LIN {X 0,Y 584.034,Z 289.728,A -85,B 0,C 180,E1 27907.179,E2 27907.179} C_VEL
LIN {X 0,Y 584.025,Z 289.73,A -85,B 0,C 180,E1 27903.828,E2 27903.828} C_VEL
LIN {X 0,Y 584.048,Z 289.73,A -85,B 0,C 180,E1 27900.883,E2 27900.883} C_VEL
LIN {X 0,Y 584.013,Z 289.73,A -85,B 0,C 180,E1 27897.645,E2 27897.645} C_VEL
LIN {X 0,Y 584.073,Z 289.731,A -85,B 0,C 180,E1 27894.597,E2 27894.597} C_VEL
LIN {X 0,Y 584.017,Z 289.728,A -85,B 0,C 180,E1 27891.533,E2 27891.533} C_VEL
LIN {X 0,Y 584.09,Z 289.732,A -85,B 0,C 180,E1 27888.446,E2 27888.446} C_VEL
LIN {X 0,Y 584.053,Z 289.731,A -85,B 0,C 180,E1 27886.743,E2 27886.743} C_VEL
LIN {X 0,Y 583.114,Z 289.855,A -85,B 0,C 180,E1 27885.987,E2 27885.987} C_VEL
LIN {X 0,Y 576.625,Z 290.656,A -85,B 0,C 180,E1 27883.866,E2 27883.866} C_VEL
LIN {X 0,Y 576.086,Z 290.719,A -85,B 0,C 180,E1 27883.314,E2 27883.314} C_VEL
LIN {X 0,Y 576.152,Z 290.716,A -85,B 0,C 180,E1 27880.146,E2 27880.146} C_VEL
LIN {X 0,Y 576.097,Z 290.719,A -85,B 0,C 180,E1 27877.014,E2 27877.014} C_VEL
LIN {X 0,Y 576.121,Z 290.717,A -85,B 0,C 180,E1 27873.733,E2 27873.733} C_VEL
LIN {X 0,Y 576.119,Z 290.718,A -85,B 0,C 180,E1 27870.698,E2 27870.698} C_VEL
LIN {X 0,Y 576.11,Z 290.716,A -85,B 0,C 180,E1 27867.451,E2 27867.451} C_VEL
LIN {X 0,Y 576.157,Z 290.721,A -85,B 0,C 180,E1 27864.306,E2 27864.306} C_VEL
LIN {X 0,Y 576.107,Z 290.717,A -85,B 0,C 180,E1 27861.077,E2 27861.077} C_VEL
LIN {X 0,Y 576.158,Z 290.714,A -85,B 0,C 180,E1 27857.809,E2 27857.809} C_VEL
LIN {X 0,Y 576.125,Z 290.717,A -85,B 0,C 180,E1 27854.638,E2 27854.638} C_VEL
LIN {X 0,Y 576.124,Z 290.716,A -85,B 0,C 180,E1 27851.259,E2 27851.259} C_VEL
LIN {X 0,Y 576.159,Z 290.714,A -85,B 0,C 180,E1 27848.013,E2 27848.013} C_VEL
LIN {X 0,Y 576.122,Z 290.716,A -85,B 0,C 180,E1 27844.817,E2 27844.817} C_VEL
LIN {X 0,Y 576.157,Z 290.709,A -85,B 0,C 180,E1 27841.561,E2 27841.561} C_VEL
LIN {X 0,Y 576.149,Z 290.712,A -85,B 0,C 180,E1 27838.278,E2 27838.278} C_VEL
LIN {X 0,Y 576.195,Z 290.958,A -85,B 0,C 180,E1 27837.573,E2 27837.573} C_VEL
LIN {X 0,Y 578.029,Z 297.635,A -85,B 0,C 180,E1 27836.802,E2 27836.802} C_VEL
LIN {X 0,Y 577.51,Z 328.552,A -85,B 0,C 180,E1 27834.007,E2 27834.007} C_VEL
LIN {X 0,Y 577.497,Z 334.474,A -85,B 0,C 180,E1 27833.515,E2 27833.515} C_VEL
LIN {X 0,Y 578.386,Z 340.749,A -85,B 0,C 180,E1 27833.384,E2 27833.384} C_VEL
LIN {X 0,Y 577.84,Z 542.427,A -85,B 0,C 180,E1 27830.729,E2 27830.729} C_VEL
LIN {X 0,Y 577.687,Z 561.472,A -85,B 0,C 180,E1 27830.287,E2 27830.287} C_VEL
LIN {X 0,Y 577.482,Z 579.605,A -85,B 0,C 180,E1 27829.679,E2 27829.679} C_VEL
LIN {X 0,Y 577.264,Z 597.202,A -85,B 0,C 180,E1 27828.898,E2 27828.898} C_VEL
LIN {X 0,Y 577.039,Z 613.981,A -85,B 0,C 180,E1 27827.959,E2 27827.959} C_VEL
LIN {X 0,Y 576.792,Z 630.391,A -85,B 0,C 180,E1 27826.827,E2 27826.827} C_VEL
LIN {X 0,Y 576.559,Z 645.743,A -85,B 0,C 180,E1 27825.541,E2 27825.541} C_VEL
LIN {X 0,Y 576.356,Z 659.744,A -85,B 0,C 180,E1 27824.128,E2 27824.128} C_VEL
LIN {X 0,Y 576.203,Z 672.121,A -85,B 0,C 180,E1 27822.629,E2 27822.629} C_VEL
LIN {X 0,Y 576.085,Z 683.222,A -85,B 0,C 180,E1 27821.006,E2 27821.006} C_VEL
LIN {X 0,Y 576.006,Z 692.795,A -85,B 0,C 180,E1 27819.29,E2 27819.29} C_VEL
LIN {X 0,Y 575.956,Z 700.403,A -85,B 0,C 180,E1 27817.581,E2 27817.581} C_VEL
LIN {X 0,Y 575.92,Z 706.58,A -85,B 0,C 180,E1 27815.779,E2 27815.779} C_VEL
LIN {X 0,Y 575.92,Z 710.989,A -85,B 0,C 180,E1 27813.982,E2 27813.982} C_VEL
LIN {X 0,Y 575.917,Z 713.852,A -85,B 0,C 180,E1 27812.089,E2 27812.089} C_VEL
LIN {X 0,Y 575.911,Z 714.951,A -85,B 0,C 180,E1 27810.199,E2 27810.199} C_VEL
LIN {X 0,Y 575.913,Z 714.311,A -85,B 0,C 180,E1 27808.309,E2 27808.309} C_VEL
LIN {X 0,Y 575.909,Z 711.917,A -85,B 0,C 180,E1 27806.417,E2 27806.417} C_VEL
LIN {X 0,Y 575.922,Z 707.958,A -85,B 0,C 180,E1 27804.621,E2 27804.621} C_VEL
LIN {X 0,Y 575.945,Z 702.275,A -85,B 0,C 180,E1 27802.82,E2 27802.82} C_VEL
LIN {X 0,Y 575.981,Z 695.171,A -85,B 0,C 180,E1 27801.113,E2 27801.113} C_VEL
LIN {X 0,Y 576.057,Z 686.195,A -85,B 0,C 180,E1 27799.398,E2 27799.398} C_VEL
LIN {X 0,Y 576.164,Z 675.759,A -85,B 0,C 180,E1 27797.777,E2 27797.777} C_VEL
LIN {X 0,Y 576.31,Z 663.875,A -85,B 0,C 180,E1 27796.25,E2 27796.25} C_VEL
LIN {X 0,Y 576.497,Z 650.514,A -85,B 0,C 180,E1 27794.818,E2 27794.818} C_VEL
LIN {X 0,Y 576.72,Z 635.525,A -85,B 0,C 180,E1 27793.482,E2 27793.482} C_VEL
LIN {X 0,Y 576.962,Z 619.334,A -85,B 0,C 180,E1 27792.294,E2 27792.294} C_VEL
LIN {X 0,Y 577.183,Z 602.928,A -85,B 0,C 180,E1 27791.309,E2 27791.309} C_VEL
LIN {X 0,Y 577.431,Z 584.941,A -85,B 0,C 180,E1 27790.448,E2 27790.448} C_VEL
LIN {X 0,Y 577.637,Z 566.861,A -85,B 0,C 180,E1 27789.786,E2 27789.786} C_VEL
LIN {X 0,Y 577.801,Z 548.295,A -85,B 0,C 180,E1 27789.299,E2 27789.299} C_VEL
LIN {X 0,Y 577.907,Z 527.535,A -85,B 0,C 180,E1 27788.962,E2 27788.962} C_VEL
LIN {X 0,Y 578.217,Z 338.32,A -85,B 0,C 180,E1 27786.486,E2 27786.486} C_VEL
LIN {X 0,Y 577.47,Z 334.235,A -85,B 0,C 180,E1 27786.384,E2 27786.384} C_VEL
LIN {X 0,Y 577.872,Z 304.731,A -85,B 0,C 180,E1 27783.764,E2 27783.764} C_VEL
LIN {X 0,Y 577.859,Z 296.714,A -85,B 0,C 180,E1 27783.012,E2 27783.012} C_VEL
LIN {X 0,Y 576.195,Z 290.995,A -85,B 0,C 180,E1 27782.343,E2 27782.343} C_VEL
LIN {X 0,Y 576.146,Z 290.717,A -85,B 0,C 180,E1 27780.7,E2 27780.7} C_VEL
LIN {X 0,Y 576.133,Z 290.719,A -85,B 0,C 180,E1 27777.321,E2 27777.321} C_VEL
LIN {X 0,Y 576.154,Z 290.714,A -85,B 0,C 180,E1 27774.088,E2 27774.088} C_VEL
LIN {X 0,Y 576.124,Z 290.711,A -85,B 0,C 180,E1 27770.875,E2 27770.875} C_VEL
LIN {X 0,Y 576.153,Z 290.716,A -85,B 0,C 180,E1 27767.671,E2 27767.671} C_VEL
LIN {X 0,Y 576.149,Z 290.711,A -85,B 0,C 180,E1 27764.359,E2 27764.359} C_VEL
LIN {X 0,Y 576.119,Z 290.717,A -85,B 0,C 180,E1 27761.129,E2 27761.129} C_VEL
LIN {X 0,Y 576.161,Z 290.716,A -85,B 0,C 180,E1 27757.903,E2 27757.903} C_VEL
LIN {X 0,Y 576.111,Z 290.715,A -85,B 0,C 180,E1 27754.699,E2 27754.699} C_VEL
LIN {X 0,Y 576.145,Z 290.72,A -85,B 0,C 180,E1 27751.491,E2 27751.491} C_VEL
LIN {X 0,Y 576.118,Z 290.715,A -85,B 0,C 180,E1 27748.373,E2 27748.373} C_VEL
LIN {X 0,Y 576.107,Z 290.716,A -85,B 0,C 180,E1 27745.052,E2 27745.052} C_VEL
LIN {X 0,Y 576.151,Z 290.716,A -85,B 0,C 180,E1 27741.908,E2 27741.908} C_VEL
LIN {X 0,Y 576.091,Z 290.717,A -85,B 0,C 180,E1 27738.729,E2 27738.729} C_VEL
LIN {X 0,Y 576.158,Z 290.719,A -85,B 0,C 180,E1 27735.604,E2 27735.604} C_VEL
LIN {X 0,Y 576.085,Z 290.719,A -85,B 0,C 180,E1 27732.53,E2 27732.53} C_VEL
LIN {X 0,Y 576.138,Z 290.717,A -85,B 0,C 180,E1 27729.389,E2 27729.389} C_VEL
LIN {X 0,Y 576.083,Z 290.72,A -85,B 0,C 180,E1 27726.378,E2 27726.378} C_VEL
LIN {X 0,Y 576.113,Z 290.717,A -85,B 0,C 180,E1 27723.184,E2 27723.184} C_VEL
LIN {X 0,Y 576.078,Z 290.721,A -85,B 0,C 180,E1 27720.199,E2 27720.199} C_VEL
LIN {X 0,Y 576.086,Z 290.718,A -85,B 0,C 180,E1 27716.816,E2 27716.816} C_VEL
LIN {X 0,Y 576.111,Z 290.721,A -85,B 0,C 180,E1 27713.823,E2 27713.823} C_VEL
LIN {X 0,Y 576.086,Z 290.719,A -85,B 0,C 180,E1 27710.611,E2 27710.611} C_VEL
LIN {X 0,Y 576.154,Z 290.718,A -85,B 0,C 180,E1 27707.472,E2 27707.472} C_VEL
LIN {X 0,Y 576.089,Z 290.719,A -85,B 0,C 180,E1 27704.291,E2 27704.291} C_VEL
LIN {X 0,Y 576.153,Z 290.716,A -85,B 0,C 180,E1 27701.169,E2 27701.169} C_VEL
LIN {X 0,Y 576.099,Z 290.719,A -85,B 0,C 180,E1 27698.09,E2 27698.09} C_VEL
LIN {X 0,Y 576.131,Z 290.716,A -85,B 0,C 180,E1 27694.838,E2 27694.838} C_VEL
LIN {X 0,Y 576.123,Z 290.718,A -85,B 0,C 180,E1 27691.72,E2 27691.72} C_VEL
LIN {X 0,Y 576.11,Z 290.716,A -85,B 0,C 180,E1 27688.39,E2 27688.39} C_VEL
LIN {X 0,Y 576.16,Z 290.71,A -85,B 0,C 180,E1 27685.166,E2 27685.166} C_VEL
LIN {X 0,Y 576.113,Z 290.716,A -85,B 0,C 180,E1 27681.967,E2 27681.967} C_VEL
LIN {X 0,Y 576.149,Z 290.705,A -85,B 0,C 180,E1 27678.713,E2 27678.713} C_VEL
LIN {X 0,Y 576.145,Z 290.721,A -85,B 0,C 180,E1 27675.484,E2 27675.484} C_VEL
LIN {X 0,Y 576.123,Z 290.716,A -85,B 0,C 180,E1 27672.179,E2 27672.179} C_VEL
LIN {X 0,Y 576.158,Z 290.717,A -85,B 0,C 180,E1 27668.972,E2 27668.972} C_VEL
LIN {X 0,Y 576.132,Z 290.724,A -85,B 0,C 180,E1 27665.669,E2 27665.669} C_VEL
LIN {X 0,Y 576.212,Z 291.106,A -85,B 0,C 180,E1 27665.297,E2 27665.297} C_VEL
LIN {X 0,Y 580.102,Z 300.579,A -85,B 0,C 180,E1 27664.425,E2 27664.425} C_VEL
LIN {X 0,Y 579.434,Z 352.01,A -85,B 0,C 180,E1 27661.407,E2 27661.407} C_VEL
LIN {X 0,Y 579.088,Z 391.09,A -85,B 0,C 180,E1 27659.196,E2 27659.196} C_VEL
LIN {X 0,Y 579.657,Z 397.448,A -85,B 0,C 180,E1 27659.075,E2 27659.075} C_VEL
LIN {X 0,Y 578.923,Z 632.13,A -85,B 0,C 180,E1 27655.9,E2 27655.9} C_VEL
LIN {X 0,Y 578.771,Z 658.638,A -85,B 0,C 180,E1 27655.484,E2 27655.484} C_VEL
LIN {X 0,Y 578.549,Z 678.904,A -85,B 0,C 180,E1 27654.981,E2 27654.981} C_VEL
LIN {X 0,Y 578.317,Z 698.879,A -85,B 0,C 180,E1 27654.297,E2 27654.297} C_VEL
LIN {X 0,Y 578.011,Z 718.11,A -85,B 0,C 180,E1 27653.444,E2 27653.444} C_VEL
LIN {X 0,Y 577.68,Z 736.382,A -85,B 0,C 180,E1 27652.444,E2 27652.444} C_VEL
LIN {X 0,Y 577.339,Z 754.925,A -85,B 0,C 180,E1 27651.22,E2 27651.22} C_VEL
LIN {X 0,Y 577.023,Z 772.23,A -85,B 0,C 180,E1 27649.853,E2 27649.853} C_VEL
LIN {X 0,Y 576.738,Z 788.212,A -85,B 0,C 180,E1 27648.363,E2 27648.363} C_VEL
LIN {X 0,Y 576.505,Z 802.557,A -85,B 0,C 180,E1 27646.793,E2 27646.793} C_VEL
LIN {X 0,Y 576.304,Z 815.862,A -85,B 0,C 180,E1 27645.084,E2 27645.084} C_VEL
LIN {X 0,Y 576.155,Z 828.148,A -85,B 0,C 180,E1 27643.206,E2 27643.206} C_VEL
LIN {X 0,Y 576.041,Z 838.568,A -85,B 0,C 180,E1 27641.277,E2 27641.277} C_VEL
LIN {X 0,Y 575.978,Z 846.875,A -85,B 0,C 180,E1 27639.391,E2 27639.391} C_VEL
LIN {X 0,Y 575.935,Z 853.9,A -85,B 0,C 180,E1 27637.381,E2 27637.381} C_VEL
LIN {X 0,Y 575.916,Z 859.144,A -85,B 0,C 180,E1 27635.379,E2 27635.379} C_VEL
LIN {X 0,Y 575.909,Z 862.738,A -85,B 0,C 180,E1 27633.363,E2 27633.363} C_VEL
LIN {X 0,Y 575.905,Z 864.64,A -85,B 0,C 180,E1 27631.293,E2 27631.293} C_VEL
LIN {X 0,Y 575.904,Z 864.851,A -85,B 0,C 180,E1 27629.304,E2 27629.304} C_VEL
LIN {X 0,Y 575.912,Z 863.392,A -85,B 0,C 180,E1 27627.214,E2 27627.214} C_VEL
LIN {X 0,Y 575.921,Z 860.169,A -85,B 0,C 180,E1 27625.12,E2 27625.12} C_VEL
LIN {X 0,Y 575.935,Z 855.414,A -85,B 0,C 180,E1 27623.12,E2 27623.12} C_VEL
LIN {X 0,Y 575.961,Z 848.851,A -85,B 0,C 180,E1 27621.112,E2 27621.112} C_VEL
LIN {X 0,Y 576.009,Z 840.796,A -85,B 0,C 180,E1 27619.195,E2 27619.195} C_VEL
LIN {X 0,Y 576.104,Z 830.84,A -85,B 0,C 180,E1 27617.267,E2 27617.267} C_VEL
LIN {X 0,Y 576.251,Z 819.393,A -85,B 0,C 180,E1 27615.429,E2 27615.429} C_VEL
LIN {X 0,Y 576.434,Z 806.45,A -85,B 0,C 180,E1 27613.681,E2 27613.681} C_VEL
LIN {X 0,Y 576.677,Z 791.978,A -85,B 0,C 180,E1 27612.024,E2 27612.024} C_VEL
LIN {X 0,Y 576.958,Z 776.494,A -85,B 0,C 180,E1 27610.517,E2 27610.517} C_VEL
LIN {X 0,Y 577.285,Z 759.282,A -85,B 0,C 180,E1 27609.097,E2 27609.097} C_VEL
LIN {X 0,Y 577.625,Z 740.912,A -85,B 0,C 180,E1 27607.831,E2 27607.831} C_VEL
LIN {X 0,Y 577.928,Z 722.295,A -85,B 0,C 180,E1 27606.769,E2 27606.769} C_VEL
LIN {X 0,Y 578.217,Z 703.186,A -85,B 0,C 180,E1 27605.881,E2 27605.881} C_VEL
LIN {X 0,Y 578.509,Z 682.546,A -85,B 0,C 180,E1 27605.132,E2 27605.132} C_VEL
LIN {X 0,Y 578.751,Z 662.256,A -85,B 0,C 180,E1 27604.592,E2 27604.592} C_VEL
LIN {X 0,Y 578.896,Z 641.479,A -85,B 0,C 180,E1 27604.225,E2 27604.225} C_VEL
LIN {X 0,Y 579.633,Z 403.425,A -85,B 0,C 180,E1 27601.007,E2 27601.007} C_VEL
LIN {X 0,Y 579.421,Z 393.381,A -85,B 0,C 180,E1 27600.856,E2 27600.856} C_VEL
LIN {X 0,Y 578.998,Z 389.593,A -85,B 0,C 180,E1 27600.745,E2 27600.745} C_VEL
LIN {X 0,Y 579.691,Z 333.246,A -85,B 0,C 180,E1 27597.504,E2 27597.504} C_VEL
LIN {X 0,Y 580.101,Z 300.579,A -85,B 0,C 180,E1 27595.575,E2 27595.575} C_VEL
LIN {X 0,Y 576.219,Z 291.141,A -85,B 0,C 180,E1 27594.704,E2 27594.704} C_VEL
LIN {X 0,Y 576.132,Z 290.723,A -85,B 0,C 180,E1 27594.311,E2 27594.311} C_VEL
LIN {X 0,Y 576.158,Z 290.717,A -85,B 0,C 180,E1 27591.028,E2 27591.028} C_VEL
LIN {X 0,Y 576.124,Z 290.716,A -85,B 0,C 180,E1 27587.808,E2 27587.808} C_VEL
LIN {X 0,Y 576.144,Z 290.721,A -85,B 0,C 180,E1 27584.501,E2 27584.501} C_VEL
LIN {X 0,Y 576.152,Z 290.704,A -85,B 0,C 180,E1 27581.258,E2 27581.258} C_VEL
LIN {X 0,Y 576.114,Z 290.716,A -85,B 0,C 180,E1 27578.01,E2 27578.01} C_VEL
LIN {X 0,Y 576.16,Z 290.71,A -85,B 0,C 180,E1 27574.816,E2 27574.816} C_VEL
LIN {X 0,Y 576.11,Z 290.716,A -85,B 0,C 180,E1 27571.61,E2 27571.61} C_VEL
LIN {X 0,Y 576.125,Z 290.718,A -85,B 0,C 180,E1 27568.28,E2 27568.28} C_VEL
LIN {X 0,Y 576.132,Z 290.716,A -85,B 0,C 180,E1 27565.162,E2 27565.162} C_VEL
LIN {X 0,Y 576.101,Z 290.719,A -85,B 0,C 180,E1 27561.91,E2 27561.91} C_VEL
LIN {X 0,Y 576.161,Z 290.717,A -85,B 0,C 180,E1 27558.726,E2 27558.726} C_VEL
LIN {X 0,Y 576.092,Z 290.719,A -85,B 0,C 180,E1 27555.587,E2 27555.587} C_VEL
LIN {X 0,Y 576.146,Z 290.721,A -85,B 0,C 180,E1 27552.427,E2 27552.427} C_VEL
LIN {X 0,Y 576.088,Z 290.718,A -85,B 0,C 180,E1 27549.389,E2 27549.389} C_VEL
LIN {X 0,Y 576.117,Z 290.721,A -85,B 0,C 180,E1 27546.177,E2 27546.177} C_VEL
LIN {X 0,Y 576.088,Z 290.718,A -85,B 0,C 180,E1 27543.184,E2 27543.184} C_VEL
LIN {X 0,Y 576.084,Z 290.721,A -85,B 0,C 180,E1 27539.801,E2 27539.801} C_VEL
LIN {X 0,Y 576.107,Z 290.718,A -85,B 0,C 180,E1 27536.816,E2 27536.816} C_VEL
LIN {X 0,Y 576.078,Z 290.72,A -85,B 0,C 180,E1 27533.622,E2 27533.622} C_VEL
LIN {X 0,Y 576.116,Z 290.717,A -85,B 0,C 180,E1 27530.711,E2 27530.711} C_VEL
LIN {X 0,Y 576.084,Z 290.719,A -85,B 0,C 180,E1 27527.572,E2 27527.572} C_VEL
LIN {X 0,Y 576.144,Z 290.717,A -85,B 0,C 180,E1 27524.499,E2 27524.499} C_VEL
LIN {X 0,Y 576.086,Z 290.719,A -85,B 0,C 180,E1 27523.314,E2 27523.314} C_VEL
LIN {X 0,Y 575.12,Z 290.849,A -85,B 0,C 180,E1 27522.548,E2 27522.548} C_VEL
LIN {X 0,Y 568.65,Z 291.651,A -85,B 0,C 180,E1 27520.342,E2 27520.342} C_VEL
LIN {X 0,Y 568.18,Z 291.705,A -85,B 0,C 180,E1 27519.837,E2 27519.837} C_VEL
LIN {X 0,Y 568.172,Z 291.709,A -85,B 0,C 180,E1 27516.784,E2 27516.784} C_VEL
LIN {X 0,Y 568.163,Z 291.707,A -85,B 0,C 180,E1 27513.449,E2 27513.449} C_VEL
LIN {X 0,Y 568.223,Z 291.705,A -85,B 0,C 180,E1 27510.25,E2 27510.25} C_VEL
LIN {X 0,Y 568.163,Z 291.707,A -85,B 0,C 180,E1 27507.058,E2 27507.058} C_VEL
LIN {X 0,Y 568.217,Z 291.704,A -85,B 0,C 180,E1 27503.867,E2 27503.867} C_VEL
LIN {X 0,Y 568.181,Z 291.708,A -85,B 0,C 180,E1 27500.69,E2 27500.69} C_VEL
LIN {X 0,Y 568.182,Z 291.705,A -85,B 0,C 180,E1 27497.351,E2 27497.351} C_VEL
LIN {X 0,Y 568.22,Z 291.697,A -85,B 0,C 180,E1 27494.116,E2 27494.116} C_VEL
LIN {X 0,Y 568.178,Z 291.707,A -85,B 0,C 180,E1 27490.89,E2 27490.89} C_VEL
LIN {X 0,Y 568.217,Z 291.702,A -85,B 0,C 180,E1 27487.631,E2 27487.631} C_VEL
LIN {X 0,Y 568.213,Z 291.7,A -85,B 0,C 180,E1 27484.269,E2 27484.269} C_VEL
LIN {X 0,Y 568.188,Z 291.7,A -85,B 0,C 180,E1 27481.019,E2 27481.019} C_VEL
LIN {X 0,Y 568.24,Z 291.869,A -85,B 0,C 180,E1 27477.992,E2 27477.992} C_VEL
LIN {X 0,Y 570.698,Z 300.422,A -85,B 0,C 180,E1 27476.985,E2 27476.985} C_VEL
LIN {X 0,Y 569.938,Z 334.437,A -85,B 0,C 180,E1 27473.858,E2 27473.858} C_VEL
LIN {X 0,Y 571.042,Z 341.802,A -85,B 0,C 180,E1 27473.69,E2 27473.69} C_VEL
LIN {X 0,Y 570.357,Z 542.461,A -85,B 0,C 180,E1 27471.014,E2 27471.014} C_VEL
LIN {X 0,Y 570.168,Z 561.439,A -85,B 0,C 180,E1 27470.568,E2 27470.568} C_VEL
LIN {X 0,Y 569.912,Z 579.619,A -85,B 0,C 180,E1 27469.951,E2 27469.951} C_VEL
LIN {X 0,Y 569.638,Z 597.212,A -85,B 0,C 180,E1 27469.161,E2 27469.161} C_VEL
LIN {X 0,Y 569.346,Z 613.904,A -85,B 0,C 180,E1 27468.215,E2 27468.215} C_VEL
LIN {X 0,Y 569.043,Z 630.096,A -85,B 0,C 180,E1 27467.087,E2 27467.087} C_VEL
LIN {X 0,Y 568.755,Z 645.194,A -85,B 0,C 180,E1 27465.812,E2 27465.812} C_VEL
LIN {X 0,Y 568.513,Z 658.551,A -85,B 0,C 180,E1 27464.462,E2 27464.462} C_VEL
LIN {X 0,Y 568.303,Z 671.355,A -85,B 0,C 180,E1 27462.911,E2 27462.911} C_VEL
LIN {X 0,Y 568.139,Z 682.59,A -85,B 0,C 180,E1 27461.265,E2 27461.265} C_VEL
LIN {X 0,Y 568.028,Z 692.284,A -85,B 0,C 180,E1 27459.524,E2 27459.524} C_VEL
LIN {X 0,Y 567.964,Z 700.001,A -85,B 0,C 180,E1 27457.79,E2 27457.79} C_VEL
LIN {X 0,Y 567.93,Z 706.281,A -85,B 0,C 180,E1 27455.962,E2 27455.962} C_VEL
LIN {X 0,Y 567.92,Z 710.991,A -85,B 0,C 180,E1 27454.038,E2 27454.038} C_VEL
LIN {X 0,Y 567.917,Z 713.854,A -85,B 0,C 180,E1 27452.119,E2 27452.119} C_VEL
LIN {X 0,Y 567.911,Z 714.951,A -85,B 0,C 180,E1 27450.202,E2 27450.202} C_VEL
LIN {X 0,Y 567.913,Z 714.31,A -85,B 0,C 180,E1 27448.285,E2 27448.285} C_VEL
LIN {X 0,Y 567.911,Z 711.916,A -85,B 0,C 180,E1 27446.366,E2 27446.366} C_VEL
LIN {X 0,Y 567.926,Z 707.956,A -85,B 0,C 180,E1 27444.545,E2 27444.545} C_VEL
LIN {X 0,Y 567.952,Z 702.272,A -85,B 0,C 180,E1 27442.718,E2 27442.718} C_VEL
LIN {X 0,Y 568.01,Z 694.957,A -85,B 0,C 180,E1 27440.94,E2 27440.94} C_VEL
LIN {X 0,Y 568.097,Z 686.193,A -85,B 0,C 180,E1 27439.248,E2 27439.248} C_VEL
LIN {X 0,Y 568.244,Z 675.52,A -85,B 0,C 180,E1 27437.57,E2 27437.57} C_VEL
LIN {X 0,Y 568.423,Z 663.87,A -85,B 0,C 180,E1 27436.056,E2 27436.056} C_VEL
LIN {X 0,Y 568.659,Z 650.506,A -85,B 0,C 180,E1 27434.604,E2 27434.604} C_VEL
LIN {X 0,Y 568.942,Z 635.518,A -85,B 0,C 180,E1 27433.25,E2 27433.25} C_VEL
LIN {X 0,Y 569.246,Z 619.329,A -85,B 0,C 180,E1 27432.046,E2 27432.046} C_VEL
LIN {X 0,Y 569.532,Z 602.921,A -85,B 0,C 180,E1 27431.048,E2 27431.048} C_VEL
LIN {X 0,Y 569.835,Z 585.631,A -85,B 0,C 180,E1 27430.206,E2 27430.206} C_VEL
LIN {X 0,Y 570.095,Z 567.459,A -85,B 0,C 180,E1 27429.526,E2 27429.526} C_VEL
LIN {X 0,Y 570.302,Z 548.912,A -85,B 0,C 180,E1 27429.028,E2 27429.028} C_VEL
LIN {X 0,Y 570.433,Z 528.629,A -85,B 0,C 180,E1 27428.688,E2 27428.688} C_VEL
LIN {X 0,Y 570.885,Z 339.627,A -85,B 0,C 180,E1 27426.184,E2 27426.184} C_VEL
LIN {X 0,Y 569.914,Z 334.093,A -85,B 0,C 180,E1 27426.032,E2 27426.032} C_VEL
LIN {X 0,Y 570.703,Z 300.17,A -85,B 0,C 180,E1 27422.903,E2 27422.903} C_VEL
LIN {X 0,Y 568.242,Z 291.898,A -85,B 0,C 180,E1 27421.922,E2 27421.922} C_VEL
LIN {X 0,Y 568.211,Z 291.697,A -85,B 0,C 180,E1 27418.611,E2 27418.611} C_VEL
LIN {X 0,Y 568.191,Z 291.705,A -85,B 0,C 180,E1 27415.265,E2 27415.265} C_VEL
LIN {X 0,Y 568.218,Z 291.702,A -85,B 0,C 180,E1 27411.986,E2 27411.986} C_VEL
LIN {X 0,Y 568.19,Z 291.704,A -85,B 0,C 180,E1 27408.709,E2 27408.709} C_VEL
LIN {X 0,Y 568.191,Z 291.705,A -85,B 0,C 180,E1 27405.311,E2 27405.311} C_VEL
LIN {X 0,Y 568.221,Z 291.704,A -85,B 0,C 180,E1 27402.052,E2 27402.052} C_VEL
LIN {X 0,Y 568.175,Z 291.705,A -85,B 0,C 180,E1 27398.78,E2 27398.78} C_VEL
LIN {X 0,Y 568.206,Z 291.708,A -85,B 0,C 180,E1 27395.5,E2 27395.5} C_VEL
LIN {X 0,Y 568.188,Z 291.704,A -85,B 0,C 180,E1 27392.341,E2 27392.341} C_VEL
LIN {X 0,Y 568.171,Z 291.706,A -85,B 0,C 180,E1 27389.059,E2 27389.059} C_VEL
LIN {X 0,Y 568.219,Z 291.705,A -85,B 0,C 180,E1 27385.874,E2 27385.874} C_VEL
LIN {X 0,Y 568.159,Z 291.707,A -85,B 0,C 180,E1 27382.669,E2 27382.669} C_VEL
LIN {X 0,Y 568.199,Z 291.707,A -85,B 0,C 180,E1 27379.426,E2 27379.426} C_VEL
LIN {X 0,Y 568.16,Z 291.707,A -85,B 0,C 180,E1 27376.354,E2 27376.354} C_VEL
LIN {X 0,Y 568.161,Z 291.708,A -85,B 0,C 180,E1 27373.018,E2 27373.018} C_VEL
LIN {X 0,Y 568.173,Z 291.707,A -85,B 0,C 180,E1 27370.033,E2 27370.033} C_VEL
LIN {X 0,Y 568.144,Z 291.709,A -85,B 0,C 180,E1 27366.772,E2 27366.772} C_VEL
LIN {X 0,Y 568.206,Z 291.708,A -85,B 0,C 180,E1 27363.632,E2 27363.632} C_VEL
LIN {X 0,Y 568.134,Z 291.71,A -85,B 0,C 180,E1 27360.504,E2 27360.504} C_VEL
LIN {X 0,Y 568.204,Z 291.705,A -85,B 0,C 180,E1 27357.378,E2 27357.378} C_VEL
LIN {X 0,Y 568.143,Z 291.709,A -85,B 0,C 180,E1 27354.243,E2 27354.243} C_VEL
LIN {X 0,Y 568.173,Z 291.707,A -85,B 0,C 180,E1 27350.989,E2 27350.989} C_VEL
LIN {X 0,Y 568.158,Z 291.709,A -85,B 0,C 180,E1 27348.015,E2 27348.015} C_VEL
LIN {X 0,Y 568.159,Z 291.708,A -85,B 0,C 180,E1 27344.656,E2 27344.656} C_VEL
LIN {X 0,Y 568.193,Z 291.708,A -85,B 0,C 180,E1 27341.64,E2 27341.64} C_VEL
LIN {X 0,Y 568.158,Z 291.707,A -85,B 0,C 180,E1 27338.42,E2 27338.42} C_VEL
LIN {X 0,Y 568.224,Z 291.706,A -85,B 0,C 180,E1 27335.222,E2 27335.222} C_VEL
LIN {X 0,Y 568.164,Z 291.706,A -85,B 0,C 180,E1 27332.055,E2 27332.055} C_VEL
LIN {X 0,Y 568.198,Z 291.703,A -85,B 0,C 180,E1 27328.781,E2 27328.781} C_VEL
LIN {X 0,Y 568.194,Z 291.709,A -85,B 0,C 180,E1 27325.607,E2 27325.607} C_VEL
LIN {X 0,Y 568.178,Z 291.703,A -85,B 0,C 180,E1 27322.361,E2 27322.361} C_VEL
LIN {X 0,Y 568.221,Z 291.697,A -85,B 0,C 180,E1 27319.167,E2 27319.167} C_VEL
LIN {X 0,Y 568.181,Z 291.708,A -85,B 0,C 180,E1 27315.886,E2 27315.886} C_VEL
LIN {X 0,Y 568.213,Z 291.703,A -85,B 0,C 180,E1 27312.644,E2 27312.644} C_VEL
LIN {X 0,Y 568.219,Z 291.7,A -85,B 0,C 180,E1 27309.264,E2 27309.264} C_VEL
LIN {X 0,Y 568.189,Z 291.725,A -85,B 0,C 180,E1 27305.956,E2 27305.956} C_VEL
LIN {X 0,Y 568.299,Z 292.358,A -85,B 0,C 180,E1 27305.739,E2 27305.739} C_VEL
LIN {X 0,Y 573.205,Z 304.206,A -85,B 0,C 180,E1 27304.675,E2 27304.675} C_VEL
LIN {X 0,Y 572.309,Z 356.956,A -85,B 0,C 180,E1 27301.549,E2 27301.549} C_VEL
LIN {X 0,Y 571.927,Z 391.105,A -85,B 0,C 180,E1 27299.597,E2 27299.597} C_VEL
LIN {X 0,Y 572.661,Z 398.211,A -85,B 0,C 180,E1 27299.454,E2 27299.454} C_VEL
LIN {X 0,Y 571.724,Z 632.462,A -85,B 0,C 180,E1 27296.246,E2 27296.246} C_VEL
LIN {X 0,Y 571.533,Z 658.799,A -85,B 0,C 180,E1 27295.827,E2 27295.827} C_VEL
LIN {X 0,Y 571.26,Z 679.227,A -85,B 0,C 180,E1 27295.312,E2 27295.312} C_VEL
LIN {X 0,Y 570.968,Z 698.877,A -85,B 0,C 180,E1 27294.63,E2 27294.63} C_VEL
LIN {X 0,Y 570.579,Z 718.114,A -85,B 0,C 180,E1 27293.768,E2 27293.768} C_VEL
LIN {X 0,Y 570.153,Z 737.04,A -85,B 0,C 180,E1 27292.717,E2 27292.717} C_VEL
LIN {X 0,Y 569.744,Z 754.928,A -85,B 0,C 180,E1 27291.516,E2 27291.516} C_VEL
LIN {X 0,Y 569.343,Z 772.232,A -85,B 0,C 180,E1 27290.133,E2 27290.133} C_VEL
LIN {X 0,Y 568.969,Z 788.436,A -85,B 0,C 180,E1 27288.599,E2 27288.599} C_VEL
LIN {X 0,Y 568.661,Z 803.058,A -85,B 0,C 180,E1 27286.97,E2 27286.97} C_VEL
LIN {X 0,Y 568.418,Z 815.863,A -85,B 0,C 180,E1 27285.298,E2 27285.298} C_VEL
LIN {X 0,Y 568.225,Z 827.928,A -85,B 0,C 180,E1 27283.43,E2 27283.43} C_VEL
LIN {X 0,Y 568.078,Z 837.883,A -85,B 0,C 180,E1 27281.575,E2 27281.575} C_VEL
LIN {X 0,Y 567.992,Z 846.469,A -85,B 0,C 180,E1 27279.627,E2 27279.627} C_VEL
LIN {X 0,Y 567.947,Z 853.597,A -85,B 0,C 180,E1 27277.587,E2 27277.587} C_VEL
LIN {X 0,Y 567.925,Z 858.73,A -85,B 0,C 180,E1 27275.658,E2 27275.658} C_VEL
LIN {X 0,Y 567.909,Z 862.558,A -85,B 0,C 180,E1 27273.533,E2 27273.533} C_VEL
LIN {X 0,Y 567.902,Z 864.507,A -85,B 0,C 180,E1 27271.513,E2 27271.513} C_VEL
LIN {X 0,Y 567.9,Z 864.896,A -85,B 0,C 180,E1 27269.496,E2 27269.496} C_VEL
LIN {X 0,Y 567.901,Z 863.728,A -85,B 0,C 180,E1 27267.477,E2 27267.477} C_VEL
LIN {X 0,Y 567.907,Z 860.972,A -85,B 0,C 180,E1 27265.456,E2 27265.456} C_VEL
LIN {X 0,Y 567.926,Z 856.483,A -85,B 0,C 180,E1 27263.429,E2 27263.429} C_VEL
LIN {X 0,Y 567.965,Z 850.267,A -85,B 0,C 180,E1 27261.394,E2 27261.394} C_VEL
LIN {X 0,Y 568.03,Z 842.181,A -85,B 0,C 180,E1 27259.349,E2 27259.349} C_VEL
LIN {X 0,Y 568.145,Z 832.569,A -85,B 0,C 180,E1 27257.396,E2 27257.396} C_VEL
LIN {X 0,Y 568.32,Z 821.497,A -85,B 0,C 180,E1 27255.533,E2 27255.533} C_VEL
LIN {X 0,Y 568.551,Z 808.943,A -85,B 0,C 180,E1 27253.763,E2 27253.763} C_VEL
LIN {X 0,Y 568.837,Z 794.891,A -85,B 0,C 180,E1 27252.086,E2 27252.086} C_VEL
LIN {X 0,Y 569.168,Z 779.848,A -85,B 0,C 180,E1 27250.556,E2 27250.556} C_VEL
LIN {X 0,Y 569.55,Z 763.302,A -85,B 0,C 180,E1 27249.123,E2 27249.123} C_VEL
LIN {X 0,Y 569.976,Z 744.963,A -85,B 0,C 180,E1 27247.789,E2 27247.789} C_VEL
LIN {X 0,Y 570.378,Z 726.292,A -85,B 0,C 180,E1 27246.662,E2 27246.662} C_VEL
LIN {X 0,Y 570.785,Z 707.828,A -85,B 0,C 180,E1 27245.747,E2 27245.747} C_VEL
LIN {X 0,Y 571.158,Z 687.897,A -85,B 0,C 180,E1 27244.964,E2 27244.964} C_VEL
LIN {X 0,Y 571.425,Z 667.643,A -85,B 0,C 180,E1 27244.371,E2 27244.371} C_VEL
LIN {X 0,Y 571.645,Z 647.244,A -85,B 0,C 180,E1 27243.965,E2 27243.965} C_VEL
LIN {X 0,Y 572.627,Z 405.206,A -85,B 0,C 180,E1 27240.643,E2 27240.643} C_VEL
LIN {X 0,Y 572.429,Z 394.559,A -85,B 0,C 180,E1 27240.481,E2 27240.481} C_VEL
LIN {X 0,Y 571.833,Z 389.593,A -85,B 0,C 180,E1 27240.342,E2 27240.342} C_VEL
LIN {X 0,Y 572.729,Z 332.228,A -85,B 0,C 180,E1 27236.998,E2 27236.998} C_VEL
LIN {X 0,Y 573.013,Z 303.541,A -85,B 0,C 180,E1 27235.271,E2 27235.271} C_VEL
LIN {X 0,Y 568.253,Z 292.129,A -85,B 0,C 180,E1 27234.229,E2 27234.229} C_VEL
LIN {X 0,Y 568.189,Z 291.704,A -85,B 0,C 180,E1 27233.873,E2 27233.873} C_VEL
LIN {X 0,Y 568.209,Z 291.699,A -85,B 0,C 180,E1 27230.564,E2 27230.564} C_VEL
LIN {X 0,Y 568.219,Z 291.704,A -85,B 0,C 180,E1 27227.203,E2 27227.203} C_VEL
LIN {X 0,Y 568.179,Z 291.707,A -85,B 0,C 180,E1 27223.969,E2 27223.969} C_VEL
LIN {X 0,Y 568.221,Z 291.7,A -85,B 0,C 180,E1 27220.679,E2 27220.679} C_VEL
LIN {X 0,Y 568.187,Z 291.702,A -85,B 0,C 180,E1 27217.475,E2 27217.475} C_VEL
LIN {X 0,Y 568.178,Z 291.708,A -85,B 0,C 180,E1 27214.15,E2 27214.15} C_VEL
LIN {X 0,Y 568.222,Z 291.703,A -85,B 0,C 180,E1 27210.918,E2 27210.918} C_VEL
LIN {X 0,Y 568.165,Z 291.705,A -85,B 0,C 180,E1 27207.683,E2 27207.683} C_VEL
LIN {X 0,Y 568.202,Z 291.708,A -85,B 0,C 180,E1 27204.426,E2 27204.426} C_VEL
LIN {X 0,Y 568.17,Z 291.706,A -85,B 0,C 180,E1 27201.363,E2 27201.363} C_VEL
LIN {X 0,Y 568.166,Z 291.707,A -85,B 0,C 180,E1 27198.042,E2 27198.042} C_VEL
LIN {X 0,Y 568.192,Z 291.706,A -85,B 0,C 180,E1 27194.971,E2 27194.971} C_VEL
LIN {X 0,Y 568.15,Z 291.709,A -85,B 0,C 180,E1 27191.779,E2 27191.779} C_VEL
LIN {X 0,Y 568.216,Z 291.705,A -85,B 0,C 180,E1 27188.602,E2 27188.602} C_VEL
LIN {X 0,Y 568.143,Z 291.709,A -85,B 0,C 180,E1 27185.453,E2 27185.453} C_VEL
LIN {X 0,Y 568.183,Z 291.708,A -85,B 0,C 180,E1 27182.219,E2 27182.219} C_VEL
LIN {X 0,Y 568.139,Z 291.71,A -85,B 0,C 180,E1 27179.294,E2 27179.294} C_VEL
LIN {X 0,Y 568.169,Z 291.709,A -85,B 0,C 180,E1 27176.064,E2 27176.064} C_VEL
LIN {X 0,Y 568.15,Z 291.71,A -85,B 0,C 180,E1 27173.025,E2 27173.025} C_VEL
LIN {X 0,Y 568.148,Z 291.709,A -85,B 0,C 180,E1 27169.651,E2 27169.651} C_VEL
LIN {X 0,Y 568.197,Z 291.709,A -85,B 0,C 180,E1 27166.568,E2 27166.568} C_VEL
LIN {X 0,Y 568.149,Z 291.708,A -85,B 0,C 180,E1 27163.435,E2 27163.435} C_VEL
LIN {X 0,Y 568.219,Z 291.704,A -85,B 0,C 180,E1 27160.254,E2 27160.254} C_VEL
LIN {X 0,Y 568.18,Z 291.705,A -85,B 0,C 180,E1 27159.837,E2 27159.837} C_VEL
LIN {X 0,Y 567.152,Z 291.832,A -85,B 0,C 180,E1 27159.061,E2 27159.061} C_VEL
LIN {X 0,Y 560.801,Z 292.636,A -85,B 0,C 180,E1 27156.88,E2 27156.88} C_VEL
LIN {X 0,Y 560.282,Z 292.693,A -85,B 0,C 180,E1 27156.313,E2 27156.313} C_VEL
LIN {X 0,Y 560.219,Z 292.697,A -85,B 0,C 180,E1 27153.157,E2 27153.157} C_VEL
LIN {X 0,Y 560.271,Z 292.693,A -85,B 0,C 180,E1 27149.902,E2 27149.902} C_VEL
LIN {X 0,Y 560.236,Z 292.697,A -85,B 0,C 180,E1 27146.776,E2 27146.776} C_VEL
LIN {X 0,Y 560.238,Z 292.694,A -85,B 0,C 180,E1 27143.409,E2 27143.409} C_VEL
LIN {X 0,Y 560.286,Z 292.696,A -85,B 0,C 180,E1 27140.159,E2 27140.159} C_VEL
LIN {X 0,Y 560.236,Z 292.696,A -85,B 0,C 180,E1 27136.879,E2 27136.879} C_VEL
LIN {X 0,Y 560.263,Z 292.684,A -85,B 0,C 180,E1 27133.539,E2 27133.539} C_VEL
LIN {X 0,Y 560.279,Z 292.694,A -85,B 0,C 180,E1 27130.199,E2 27130.199} C_VEL
LIN {X 0,Y 560.243,Z 292.694,A -85,B 0,C 180,E1 27126.913,E2 27126.913} C_VEL
LIN {X 0,Y 560.28,Z 292.691,A -85,B 0,C 180,E1 27123.587,E2 27123.587} C_VEL
LIN {X 0,Y 560.279,Z 292.687,A -85,B 0,C 180,E1 27120.214,E2 27120.214} C_VEL
LIN {X 0,Y 560.305,Z 292.964,A -85,B 0,C 180,E1 27118.387,E2 27118.387} C_VEL
LIN {X 0,Y 563.388,Z 303.018,A -85,B 0,C 180,E1 27117.192,E2 27117.192} C_VEL
LIN {X 0,Y 562.6,Z 334.852,A -85,B 0,C 180,E1 27114.238,E2 27114.238} C_VEL
LIN {X 0,Y 563.916,Z 343.007,A -85,B 0,C 180,E1 27114.045,E2 27114.045} C_VEL
LIN {X 0,Y 562.881,Z 542.819,A -85,B 0,C 180,E1 27111.3,E2 27111.3} C_VEL
LIN {X 0,Y 562.657,Z 561.678,A -85,B 0,C 180,E1 27110.848,E2 27110.848} C_VEL
LIN {X 0,Y 562.355,Z 579.633,A -85,B 0,C 180,E1 27110.231,E2 27110.231} C_VEL
LIN {X 0,Y 562.024,Z 597.222,A -85,B 0,C 180,E1 27109.431,E2 27109.431} C_VEL
LIN {X 0,Y 561.663,Z 613.911,A -85,B 0,C 180,E1 27108.473,E2 27108.473} C_VEL
LIN {X 0,Y 561.306,Z 629.734,A -85,B 0,C 180,E1 27107.359,E2 27107.359} C_VEL
LIN {X 0,Y 560.965,Z 644.403,A -85,B 0,C 180,E1 27106.114,E2 27106.114} C_VEL
LIN {X 0,Y 560.675,Z 657.631,A -85,B 0,C 180,E1 27104.774,E2 27104.774} C_VEL
LIN {X 0,Y 560.424,Z 669.814,A -85,B 0,C 180,E1 27103.306,E2 27103.306} C_VEL
LIN {X 0,Y 560.219,Z 681.321,A -85,B 0,C 180,E1 27101.635,E2 27101.635} C_VEL
LIN {X 0,Y 560.081,Z 690.74,A -85,B 0,C 180,E1 27099.972,E2 27099.972} C_VEL
LIN {X 0,Y 559.997,Z 698.789,A -85,B 0,C 180,E1 27098.212,E2 27098.212} C_VEL
LIN {X 0,Y 559.939,Z 705.374,A -85,B 0,C 180,E1 27096.356,E2 27096.356} C_VEL
LIN {X 0,Y 559.921,Z 710.168,A -85,B 0,C 180,E1 27094.506,E2 27094.506} C_VEL
LIN {X 0,Y 559.907,Z 713.29,A -85,B 0,C 180,E1 27092.661,E2 27092.661} C_VEL
LIN {X 0,Y 559.915,Z 714.838,A -85,B 0,C 180,E1 27090.716,E2 27090.716} C_VEL
LIN {X 0,Y 559.909,Z 714.647,A -85,B 0,C 180,E1 27088.772,E2 27088.772} C_VEL
LIN {X 0,Y 559.914,Z 712.708,A -85,B 0,C 180,E1 27086.827,E2 27086.827} C_VEL
LIN {X 0,Y 559.923,Z 709.223,A -85,B 0,C 180,E1 27084.98,E2 27084.98} C_VEL
LIN {X 0,Y 559.952,Z 704.018,A -85,B 0,C 180,E1 27083.124,E2 27083.124} C_VEL
LIN {X 0,Y 560.005,Z 697.005,A -85,B 0,C 180,E1 27081.271,E2 27081.271} C_VEL
LIN {X 0,Y 560.112,Z 688.488,A -85,B 0,C 180,E1 27079.509,E2 27079.509} C_VEL
LIN {X 0,Y 560.259,Z 678.56,A -85,B 0,C 180,E1 27077.844,E2 27077.844} C_VEL
LIN {X 0,Y 560.47,Z 667.253,A -85,B 0,C 180,E1 27076.275,E2 27076.275} C_VEL
LIN {X 0,Y 560.738,Z 654.562,A -85,B 0,C 180,E1 27074.805,E2 27074.805} C_VEL
LIN {X 0,Y 561.057,Z 640.393,A -85,B 0,C 180,E1 27073.434,E2 27073.434} C_VEL
LIN {X 0,Y 561.423,Z 624.546,A -85,B 0,C 180,E1 27072.163,E2 27072.163} C_VEL
LIN {X 0,Y 561.79,Z 607.513,A -85,B 0,C 180,E1 27071.047,E2 27071.047} C_VEL
LIN {X 0,Y 562.163,Z 590.281,A -85,B 0,C 180,E1 27070.141,E2 27070.141} C_VEL
LIN {X 0,Y 562.487,Z 571.965,A -85,B 0,C 180,E1 27069.394,E2 27069.394} C_VEL
LIN {X 0,Y 562.753,Z 553.456,A -85,B 0,C 180,E1 27068.842,E2 27068.842} C_VEL
LIN {X 0,Y 562.941,Z 534.654,A -85,B 0,C 180,E1 27068.477,E2 27068.477} C_VEL
LIN {X 0,Y 563.774,Z 340.944,A -85,B 0,C 180,E1 27065.83,E2 27065.83} C_VEL
LIN {X 0,Y 562.571,Z 334.474,A -85,B 0,C 180,E1 27065.649,E2 27065.649} C_VEL
LIN {X 0,Y 563.375,Z 302.788,A -85,B 0,C 180,E1 27062.693,E2 27062.693} C_VEL
LIN {X 0,Y 560.303,Z 292.942,A -85,B 0,C 180,E1 27061.517,E2 27061.517} C_VEL
LIN {X 0,Y 560.278,Z 292.686,A -85,B 0,C 180,E1 27058.348,E2 27058.348} C_VEL
LIN {X 0,Y 560.25,Z 292.692,A -85,B 0,C 180,E1 27055.05,E2 27055.05} C_VEL
LIN {X 0,Y 560.277,Z 292.687,A -85,B 0,C 180,E1 27051.74,E2 27051.74} C_VEL
LIN {X 0,Y 560.277,Z 292.691,A -85,B 0,C 180,E1 27048.395,E2 27048.395} C_VEL
LIN {X 0,Y 560.243,Z 292.692,A -85,B 0,C 180,E1 27045.115,E2 27045.115} C_VEL
LIN {X 0,Y 560.283,Z 292.696,A -85,B 0,C 180,E1 27041.869,E2 27041.869} C_VEL
LIN {X 0,Y 560.245,Z 292.693,A -85,B 0,C 180,E1 27038.587,E2 27038.587} C_VEL
LIN {X 0,Y 560.241,Z 292.695,A -85,B 0,C 180,E1 27035.178,E2 27035.178} C_VEL
LIN {X 0,Y 560.285,Z 292.693,A -85,B 0,C 180,E1 27031.886,E2 27031.886} C_VEL
LIN {X 0,Y 560.226,Z 292.694,A -85,B 0,C 180,E1 27028.692,E2 27028.692} C_VEL
LIN {X 0,Y 560.263,Z 292.693,A -85,B 0,C 180,E1 27025.446,E2 27025.446} C_VEL
LIN {X 0,Y 560.233,Z 292.695,A -85,B 0,C 180,E1 27022.343,E2 27022.343} C_VEL
LIN {X 0,Y 560.219,Z 292.695,A -85,B 0,C 180,E1 27018.933,E2 27018.933} C_VEL
LIN {X 0,Y 560.28,Z 292.696,A -85,B 0,C 180,E1 27015.739,E2 27015.739} C_VEL
LIN {X 0,Y 560.208,Z 292.697,A -85,B 0,C 180,E1 27012.577,E2 27012.577} C_VEL
LIN {X 0,Y 560.254,Z 292.692,A -85,B 0,C 180,E1 27009.347,E2 27009.347} C_VEL
LIN {X 0,Y 560.206,Z 292.698,A -85,B 0,C 180,E1 27006.353,E2 27006.353} C_VEL
LIN {X 0,Y 560.223,Z 292.694,A -85,B 0,C 180,E1 27003.069,E2 27003.069} C_VEL
LIN {X 0,Y 560.208,Z 292.699,A -85,B 0,C 180,E1 27000.102,E2 27000.102} C_VEL
LIN {X 0,Y 560.203,Z 292.695,A -85,B 0,C 180,E1 26996.726,E2 26996.726} C_VEL
LIN {X 0,Y 560.269,Z 292.699,A -85,B 0,C 180,E1 26993.545,E2 26993.545} C_VEL
LIN {X 0,Y 560.205,Z 292.697,A -85,B 0,C 180,E1 26990.342,E2 26990.342} C_VEL
LIN {X 0,Y 560.256,Z 292.691,A -85,B 0,C 180,E1 26987.11,E2 26987.11} C_VEL
LIN {X 0,Y 560.219,Z 292.698,A -85,B 0,C 180,E1 26984.047,E2 26984.047} C_VEL
LIN {X 0,Y 560.225,Z 292.695,A -85,B 0,C 180,E1 26980.612,E2 26980.612} C_VEL
LIN {X 0,Y 560.275,Z 292.695,A -85,B 0,C 180,E1 26977.438,E2 26977.438} C_VEL
LIN {X 0,Y 560.223,Z 292.696,A -85,B 0,C 180,E1 26974.184,E2 26974.184} C_VEL
LIN {X 0,Y 560.274,Z 292.693,A -85,B 0,C 180,E1 26970.961,E2 26970.961} C_VEL
LIN {X 0,Y 560.243,Z 292.696,A -85,B 0,C 180,E1 26967.75,E2 26967.75} C_VEL
LIN {X 0,Y 560.238,Z 292.683,A -85,B 0,C 180,E1 26964.422,E2 26964.422} C_VEL
LIN {X 0,Y 560.283,Z 292.697,A -85,B 0,C 180,E1 26961.217,E2 26961.217} C_VEL
LIN {X 0,Y 560.238,Z 292.684,A -85,B 0,C 180,E1 26957.937,E2 26957.937} C_VEL
LIN {X 0,Y 560.268,Z 292.687,A -85,B 0,C 180,E1 26954.598,E2 26954.598} C_VEL
LIN {X 0,Y 560.28,Z 292.695,A -85,B 0,C 180,E1 26951.297,E2 26951.297} C_VEL
LIN {X 0,Y 560.247,Z 292.699,A -85,B 0,C 180,E1 26948.002,E2 26948.002} C_VEL
LIN {X 0,Y 560.282,Z 292.88,A -85,B 0,C 180,E1 26946.262,E2 26946.262} C_VEL
LIN {X 0,Y 560.934,Z 295.081,A -85,B 0,C 180,E1 26946.03,E2 26946.03} C_VEL
LIN {X 0,Y 566.263,Z 307.722,A -85,B 0,C 180,E1 26944.935,E2 26944.935} C_VEL
LIN {X 0,Y 565.204,Z 360.911,A -85,B 0,C 180,E1 26941.754,E2 26941.754} C_VEL
LIN {X 0,Y 564.776,Z 391.023,A -85,B 0,C 180,E1 26940.011,E2 26940.011} C_VEL
LIN {X 0,Y 565.688,Z 399.229,A -85,B 0,C 180,E1 26939.839,E2 26939.839} C_VEL
LIN {X 0,Y 564.542,Z 633.955,A -85,B 0,C 180,E1 26936.585,E2 26936.585} C_VEL
LIN {X 0,Y 564.314,Z 659.286,A -85,B 0,C 180,E1 26936.171,E2 26936.171} C_VEL
LIN {X 0,Y 563.973,Z 680.201,A -85,B 0,C 180,E1 26935.631,E2 26935.631} C_VEL
LIN {X 0,Y 563.598,Z 700.159,A -85,B 0,C 180,E1 26934.918,E2 26934.918} C_VEL
LIN {X 0,Y 563.149,Z 719.236,A -85,B 0,C 180,E1 26934.045,E2 26934.045} C_VEL
LIN {X 0,Y 562.629,Z 738.229,A -85,B 0,C 180,E1 26932.964,E2 26932.964} C_VEL
LIN {X 0,Y 562.143,Z 755.657,A -85,B 0,C 180,E1 26931.767,E2 26931.767} C_VEL
LIN {X 0,Y 561.656,Z 772.838,A -85,B 0,C 180,E1 26930.366,E2 26930.366} C_VEL
LIN {X 0,Y 561.186,Z 789.434,A -85,B 0,C 180,E1 26928.76,E2 26928.76} C_VEL
LIN {X 0,Y 560.814,Z 803.908,A -85,B 0,C 180,E1 26927.107,E2 26927.107} C_VEL
LIN {X 0,Y 560.519,Z 816.571,A -85,B 0,C 180,E1 26925.413,E2 26925.413} C_VEL
LIN {X 0,Y 560.286,Z 828.533,A -85,B 0,C 180,E1 26923.519,E2 26923.519} C_VEL
LIN {X 0,Y 560.111,Z 838.911,A -85,B 0,C 180,E1 26921.533,E2 26921.533} C_VEL
LIN {X 0,Y 560.008,Z 847.28,A -85,B 0,C 180,E1 26919.558,E2 26919.558} C_VEL
LIN {X 0,Y 559.953,Z 853.9,A -85,B 0,C 180,E1 26917.593,E2 26917.593} C_VEL
LIN {X 0,Y 559.922,Z 859.143,A -85,B 0,C 180,E1 26915.533,E2 26915.533} C_VEL
LIN {X 0,Y 559.909,Z 862.71,A -85,B 0,C 180,E1 26913.481,E2 26913.481} C_VEL
LIN {X 0,Y 559.904,Z 864.64,A -85,B 0,C 180,E1 26911.33,E2 26911.33} C_VEL
LIN {X 0,Y 559.905,Z 864.851,A -85,B 0,C 180,E1 26909.284,E2 26909.284} C_VEL
LIN {X 0,Y 559.914,Z 863.393,A -85,B 0,C 180,E1 26907.134,E2 26907.134} C_VEL
LIN {X 0,Y 559.924,Z 860.17,A -85,B 0,C 180,E1 26904.98,E2 26904.98} C_VEL
LIN {X 0,Y 559.947,Z 855.415,A -85,B 0,C 180,E1 26902.923,E2 26902.923} C_VEL
LIN {X 0,Y 559.995,Z 848.852,A -85,B 0,C 180,E1 26900.857,E2 26900.857} C_VEL
LIN {X 0,Y 560.079,Z 840.797,A -85,B 0,C 180,E1 26898.884,E2 26898.884} C_VEL
LIN {X 0,Y 560.235,Z 830.842,A -85,B 0,C 180,E1 26896.9,E2 26896.9} C_VEL
LIN {X 0,Y 560.454,Z 819.394,A -85,B 0,C 180,E1 26895.009,E2 26895.009} C_VEL
LIN {X 0,Y 560.746,Z 806.448,A -85,B 0,C 180,E1 26893.211,E2 26893.211} C_VEL
LIN {X 0,Y 561.103,Z 792.705,A -85,B 0,C 180,E1 26891.585,E2 26891.585} C_VEL
LIN {X 0,Y 561.533,Z 777.056,A -85,B 0,C 180,E1 26890.01,E2 26890.01} C_VEL
LIN {X 0,Y 562.026,Z 759.961,A -85,B 0,C 180,E1 26888.557,E2 26888.557} C_VEL
LIN {X 0,Y 562.532,Z 742.205,A -85,B 0,C 180,E1 26887.291,E2 26887.291} C_VEL
LIN {X 0,Y 562.996,Z 724.297,A -85,B 0,C 180,E1 26886.226,E2 26886.226} C_VEL
LIN {X 0,Y 563.466,Z 704.736,A -85,B 0,C 180,E1 26885.275,E2 26885.275} C_VEL
LIN {X 0,Y 563.906,Z 684.562,A -85,B 0,C 180,E1 26884.508,E2 26884.508} C_VEL
LIN {X 0,Y 564.273,Z 664.469,A -85,B 0,C 180,E1 26883.939,E2 26883.939} C_VEL
LIN {X 0,Y 564.493,Z 643.382,A -85,B 0,C 180,E1 26883.546,E2 26883.546} C_VEL
LIN {X 0,Y 565.655,Z 405.079,A -85,B 0,C 180,E1 26880.243,E2 26880.243} C_VEL
LIN {X 0,Y 565.443,Z 395.593,A -85,B 0,C 180,E1 26880.094,E2 26880.094} C_VEL
LIN {X 0,Y 564.695,Z 389.593,A -85,B 0,C 180,E1 26879.929,E2 26879.929} C_VEL
LIN {X 0,Y 565.793,Z 331.939,A -85,B 0,C 180,E1 26876.523,E2 26876.523} C_VEL
LIN {X 0,Y 566.206,Z 307.048,A -85,B 0,C 180,E1 26875.022,E2 26875.022} C_VEL
LIN {X 0,Y 560.335,Z 293.207,A -85,B 0,C 180,E1 26873.799,E2 26873.799} C_VEL
LIN {X 0,Y 560.268,Z 292.685,A -85,B 0,C 180,E1 26873.54,E2 26873.54} C_VEL
LIN {X 0,Y 560.247,Z 292.687,A -85,B 0,C 180,E1 26870.157,E2 26870.157} C_VEL
LIN {X 0,Y 560.279,Z 292.688,A -85,B 0,C 180,E1 26866.877,E2 26866.877} C_VEL
LIN {X 0,Y 560.252,Z 292.694,A -85,B 0,C 180,E1 26863.569,E2 26863.569} C_VEL
LIN {X 0,Y 560.244,Z 292.697,A -85,B 0,C 180,E1 26860.198,E2 26860.198} C_VEL
LIN {X 0,Y 560.283,Z 292.688,A -85,B 0,C 180,E1 26856.921,E2 26856.921} C_VEL
LIN {X 0,Y 560.233,Z 292.695,A -85,B 0,C 180,E1 26853.714,E2 26853.714} C_VEL
LIN {X 0,Y 560.265,Z 292.698,A -85,B 0,C 180,E1 26850.453,E2 26850.453} C_VEL
LIN {X 0,Y 560.247,Z 292.692,A -85,B 0,C 180,E1 26847.284,E2 26847.284} C_VEL
LIN {X 0,Y 560.228,Z 292.695,A -85,B 0,C 180,E1 26843.97,E2 26843.97} C_VEL
LIN {X 0,Y 560.282,Z 292.695,A -85,B 0,C 180,E1 26840.758,E2 26840.758} C_VEL
LIN {X 0,Y 560.216,Z 292.695,A -85,B 0,C 180,E1 26837.555,E2 26837.555} C_VEL
LIN {X 0,Y 560.25,Z 292.693,A -85,B 0,C 180,E1 26834.293,E2 26834.293} C_VEL
LIN {X 0,Y 560.222,Z 292.697,A -85,B 0,C 180,E1 26831.218,E2 26831.218} C_VEL
LIN {X 0,Y 560.217,Z 292.695,A -85,B 0,C 180,E1 26827.896,E2 26827.896} C_VEL
LIN {X 0,Y 560.248,Z 292.698,A -85,B 0,C 180,E1 26824.811,E2 26824.811} C_VEL
LIN {X 0,Y 560.201,Z 292.697,A -85,B 0,C 180,E1 26821.636,E2 26821.636} C_VEL
LIN {X 0,Y 560.271,Z 292.696,A -85,B 0,C 180,E1 26818.466,E2 26818.466} C_VEL
LIN {X 0,Y 560.198,Z 292.698,A -85,B 0,C 180,E1 26815.29,E2 26815.29} C_VEL
LIN {X 0,Y 560.241,Z 292.692,A -85,B 0,C 180,E1 26812.086,E2 26812.086} C_VEL
LIN {X 0,Y 560.215,Z 292.698,A -85,B 0,C 180,E1 26808.99,E2 26808.99} C_VEL
LIN {X 0,Y 560.215,Z 292.692,A -85,B 0,C 180,E1 26805.636,E2 26805.636} C_VEL
LIN {X 0,Y 560.256,Z 292.699,A -85,B 0,C 180,E1 26802.553,E2 26802.553} C_VEL
LIN {X 0,Y 560.213,Z 292.695,A -85,B 0,C 180,E1 26799.305,E2 26799.305} C_VEL
LIN {X 0,Y 560.282,Z 292.693,A -85,B 0,C 180,E1 26796.313,E2 26796.313} C_VEL
LIN {X 0,Y 559.276,Z 292.812,A -85,B 0,C 180,E1 26795.525,E2 26795.525} C_VEL
LIN {X 0,Y 552.789,Z 293.623,A -85,B 0,C 180,E1 26793.314,E2 26793.314} C_VEL
LIN {X 0,Y 552.299,Z 293.687,A -85,B 0,C 180,E1 26792.738,E2 26792.738} C_VEL
LIN {X 0,Y 552.291,Z 293.683,A -85,B 0,C 180,E1 26789.421,E2 26789.421} C_VEL
LIN {X 0,Y 552.343,Z 293.682,A -85,B 0,C 180,E1 26786.188,E2 26786.188} C_VEL
LIN {X 0,Y 552.293,Z 293.685,A -85,B 0,C 180,E1 26782.925,E2 26782.925} C_VEL
LIN {X 0,Y 552.319,Z 293.681,A -85,B 0,C 180,E1 26779.602,E2 26779.602} C_VEL
LIN {X 0,Y 552.327,Z 293.688,A -85,B 0,C 180,E1 26776.392,E2 26776.392} C_VEL
LIN {X 0,Y 552.3,Z 293.674,A -85,B 0,C 180,E1 26773.038,E2 26773.038} C_VEL
LIN {X 0,Y 552.341,Z 293.675,A -85,B 0,C 180,E1 26769.716,E2 26769.716} C_VEL
LIN {X 0,Y 552.33,Z 293.687,A -85,B 0,C 180,E1 26766.335,E2 26766.335} C_VEL
LIN {X 0,Y 552.311,Z 293.684,A -85,B 0,C 180,E1 26763.017,E2 26763.017} C_VEL
LIN {X 0,Y 552.342,Z 293.683,A -85,B 0,C 180,E1 26759.668,E2 26759.668} C_VEL
LIN {X 0,Y 552.352,Z 293.975,A -85,B 0,C 180,E1 26758.821,E2 26758.821} C_VEL
LIN {X 0,Y 556.072,Z 305.628,A -85,B 0,C 180,E1 26757.406,E2 26757.406} C_VEL
LIN {X 0,Y 555.276,Z 335.267,A -85,B 0,C 180,E1 26754.628,E2 26754.628} C_VEL
